# B&R Automation Studio project Parker_BMM_ST_V5_3147_V12
Automation Studio 4.2.12.129 SP

## Configuration 5AP1180_1505_parker3147

CPU 5PPC2100.BY01-000, AutomationRuntime D4.26, Build 4.1.2, Vc V4.26.8, Safety 0.0

### Task classes (Cpu.sw)
```
Cyclic#1 (cycle 2000 us, tolerance 0 us):
  tk1_in <- In_Out.tk1_in.prg
  timer <- process.timer.prg
  clamp <- process.clamp.prg
  carriage <- process.carriage.prg
  blowpin <- process.blowpin.prg
  blowpin2 <- process.blowpin2.prg
  extrlift <- process.extrlift.prg
  mc_pwr <- Motion.mc_pwr.prg [disabled]
  tk1_out <- In_Out.tk1_out.prg
  parison <- thickness.parison.prg
  robot <- process.robot.prg
  r_carriage <- Motion.r_carriage.prg [disabled]
  l_carriage <- Motion.l_carriage.prg [disabled]
  r_blowpin <- Motion.r_blowpin.prg [disabled]
  l_blowpin <- Motion.l_blowpin.prg [disabled]
  r_blowpin2 <- Motion.r_blowpin2.prg [disabled]
  l_blowpin2 <- Motion.l_blowpin2.prg [disabled]
  l_clamp <- Motion.l_clamp.prg [disabled]
  r_clamp <- Motion.r_clamp.prg [disabled]
  l_transfer <- Motion.l_transfer.prg [disabled]
  r_transfer <- Motion.r_transfer.prg [disabled]
  mc_extrlif <- Motion.mc_extrlift.prg [disabled]
  mc_thick <- Motion.mc_thick.prg [disabled]
  Trace <- screen.Trace.prg
  clean_Test <- (binary)
Cyclic#2 (cycle 10000 us, tolerance 100000 us):
  h_pwm <- Heating.h_pwm.prg
  tk2_io <- In_Out.tk2_io.prg
Cyclic#3 (cycle 4000 us, tolerance 100000 us):
  cutter <- process.cutter.prg
  cutneck <- process.cutneck.prg
  cooldef <- process.cooldef.prg
  blowdef <- process.blowdef.prg
  bdeflash <- process.bdeflash.prg
  tdeflash <- process.tdeflash.prg
  pullbottom <- process.pullbottom.prg
  inerpin <- process.inerpin.prg
  highblow <- process.highblow.prg
  lowblow <- process.lowblow.prg
  hookpin <- process.hookpin.prg
  coolpin <- process.coolpin.prg
  coolpin2 <- process.coolpin2.prg
  coolpin3 <- process.coolpin3.prg
  coolblw <- process.coolblw.prg
  coolblw2 <- process.coolblw2.prg
  coolblw3 <- process.coolblw3.prg
  robotopncl <- process.robotopncls.prg
  submold <- process.submold.prg
  pinpart <- process.pinpart.prg
  screw <- process.screw.prg
  sealer <- process.sealer.prg
  bblowpin <- process.bblowpin.prg
  support <- process.support.prg
  tonnage <- process.tonnage.prg
  autorun <- process.autorun.prg
  extru_plk <- machine.extru_plk.prg [disabled]
  extruder <- machine.extruder.prg [disabled]
  extruder_M <- machine.extruder_Mix.prg
  Acs580Ctl <- machine.Acs580Ctl.prg
  plate <- process.plate.prg
Cyclic#4 (cycle 20000 us, tolerance 200000 us):
  keyled <- screen.keyled.prg
  manual <- machine.manual.prg
  calib <- machine.calib.prg
  reset <- machine.reset.prg
  workmode <- machine.workmode.prg
  mode <- machine.mode.prg
  panel <- screen.panel.prg
  hmi_cpy <- screen.hmi_cpy.prg
  pump <- machine.pump.prg
  mac_lubr <- machine.mac_lubr.prg
  oil_accu <- machine.oil_accu.prg
  mbusMaster <- comm.mbusMaster.prg
  clean <- machine.clean.prg
  length <- process.length.prg
Cyclic#5 (cycle 500000 us, tolerance 500000 us):
  h_pid <- Heating.h_pid.prg
Cyclic#6 (cycle 30000 us, tolerance 3000000 us):
  cur_cal <- thickness.cur_cal.prg
  exchange <- thickness.exchange.prg
Cyclic#7 (cycle 50000 us, tolerance 5000000 us):
  cur_edit <- thickness.cur_edit.prg
  cur_draw <- thickness.cur_draw.prg
  pvchg <- VarChgLog.pvchg.prg
Cyclic#8 (cycle 200000 us, tolerance 30000000 us):
  spc_ctrl <- spc.spc_ctrl.prg
  trend <- Heating.trend.prg
  h_plan <- Heating.h_plan.prg
  scrshot <- screen.scrshot.prg
  hmiset <- screen.hmiset.prg
  password <- screen.password.prg
  modem <- comm.modem.prg
  vpn <- screen.vpn.prg
  recipe <- recipeMan.recipe.prg
  multsave <- recipeMan.multsave.prg
  oncesave <- recipeMan.oncesave.prg
  cur_save <- thickness.cur_save.prg
  cfg_cpy <- recipeMan.cfg_cpy.prg
  alarm <- machine.alarm.prg
  energy <- machine.energy.prg
  epl <- comm.epl.prg
DataObjects: mb_cmd <- comm.mb_cmd.dob, var_fix <- recipeMan.var_fix.dob, var_mold <- recipeMan.var_mold.dob, log_txt <- log_info.log_txt.dob, pv_chg <- VarChgLog.pv_chg.dob, cfg_dat <- recipeMan.cfg_dat.dob, Acp10sys, recName, recFix, recCurve, recMold
NcDataObjects: TransferR <- Motion.init.TransferR.dob, CarriageR <- Motion.init.CarriageR.dob, CarriageL <- Motion.init.CarriageL.dob, BlowPinR <- Motion.init.BlowPinR.dob, BlowPinL <- Motion.init.BlowPinL.dob, BlowPin2R <- Motion.init.BlowPin2R.dob, BlowPin2L <- Motion.init.BlowPin2L.dob, ThickInit <- Motion.init.ThickInit.dob, Tansfer <- Motion.para.Tansfer.dob, UpDn <- Motion.para.UpDn.dob, CarraigeLR <- Motion.para.CarraigeLR.dob, BlowPinLR <- Motion.para.BlowPinLR.dob, nCarraigeL <- Motion.para.nCarraigeLR.dob, nBlowPinLR <- Motion.para.nBlowPinLR.dob, BlowPin2LR <- Motion.para.BlowPin2LR.dob, ClampLR <- Motion.para.ClampLR.dob, acp10etxen <- Motion.acp10etxen.dob, Power <- Motion.init.Power.dob, Power1 <- Motion.para.Power.dob, ClampR <- Motion.init.ClampR.dob, ClampL <- Motion.init.ClampL.dob, ExtrLift1 <- Motion.init.ExtrLift.dob, ExtrLift2 <- Motion.para.ExtrLift.dob, ThickPara <- Motion.para.ThickPara.dob, 0804Thick, 0129_C2, gAxisPwri, gAxisPwra
VcDataObjects: visu15 <- Visu.visu15.dob
Binaries: TCData, vctcal, vccnum, vccalarm, vccovl, vcshared, visu1502, vcfile, vccstr, vccline, arial, vcctrend, vcchtml, vcgclass, vccbtn, vcrt, vccdbox, visu1503, vcclbox, simsun, vcctext, vccbmp, vcfntttf, vcalarm, vcdsint, visu1501, vccshape, vcchspot, vcmgr, vcdsloc, visvc, vccurl, vccdt, vccbar, vcpdsw, vcxml, vccscale, vcbclass, vcnet, vcpdvnc, vccddbox, vccpopup, timesbd, times, arialxsr, vccslider, vcpfar00, Role, ashwd, arconfig, iomap, User, asfw, sysconf, Acp10map, acp10cfg, vcpfmtcx, vcpk, vcpfapc, vcptelo, vcpdi815, vcpdi855, vcpdihd, vcpkat, tahomabd, arialbd, tahoma, myxh_1, myxh
Libraries: visapi, FileIO, runtime, sys_lib, standard, operator, dvframe, DataObj, Convert, brsystem, astime, asstring, AsIO, AsArLog, AsARCfg, Motorky, DRV_mbus, LoopConR, SimpFun, HydCtrl, NcGlobal, Acp10par, Acp10_MC, AsHydCon, AsEPL, Acp10man, Acp10sim, vcscrsht, powerlnk, vcresman
```

### Hardware
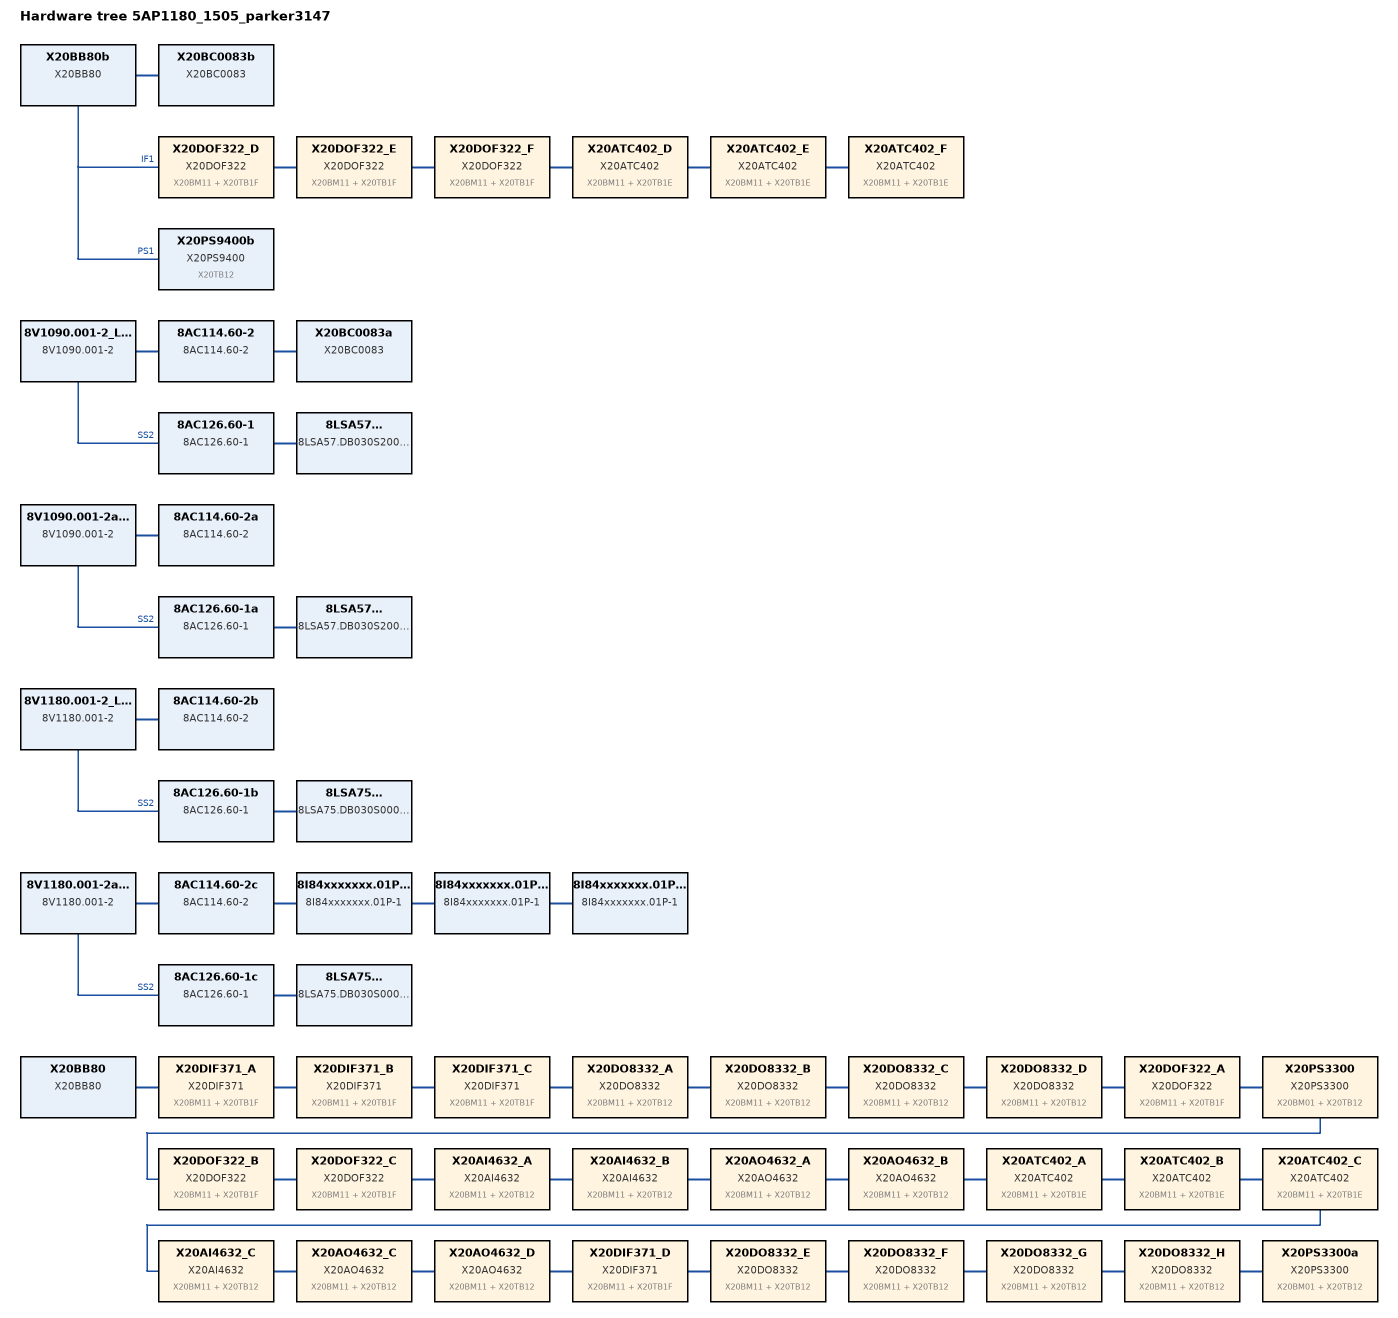
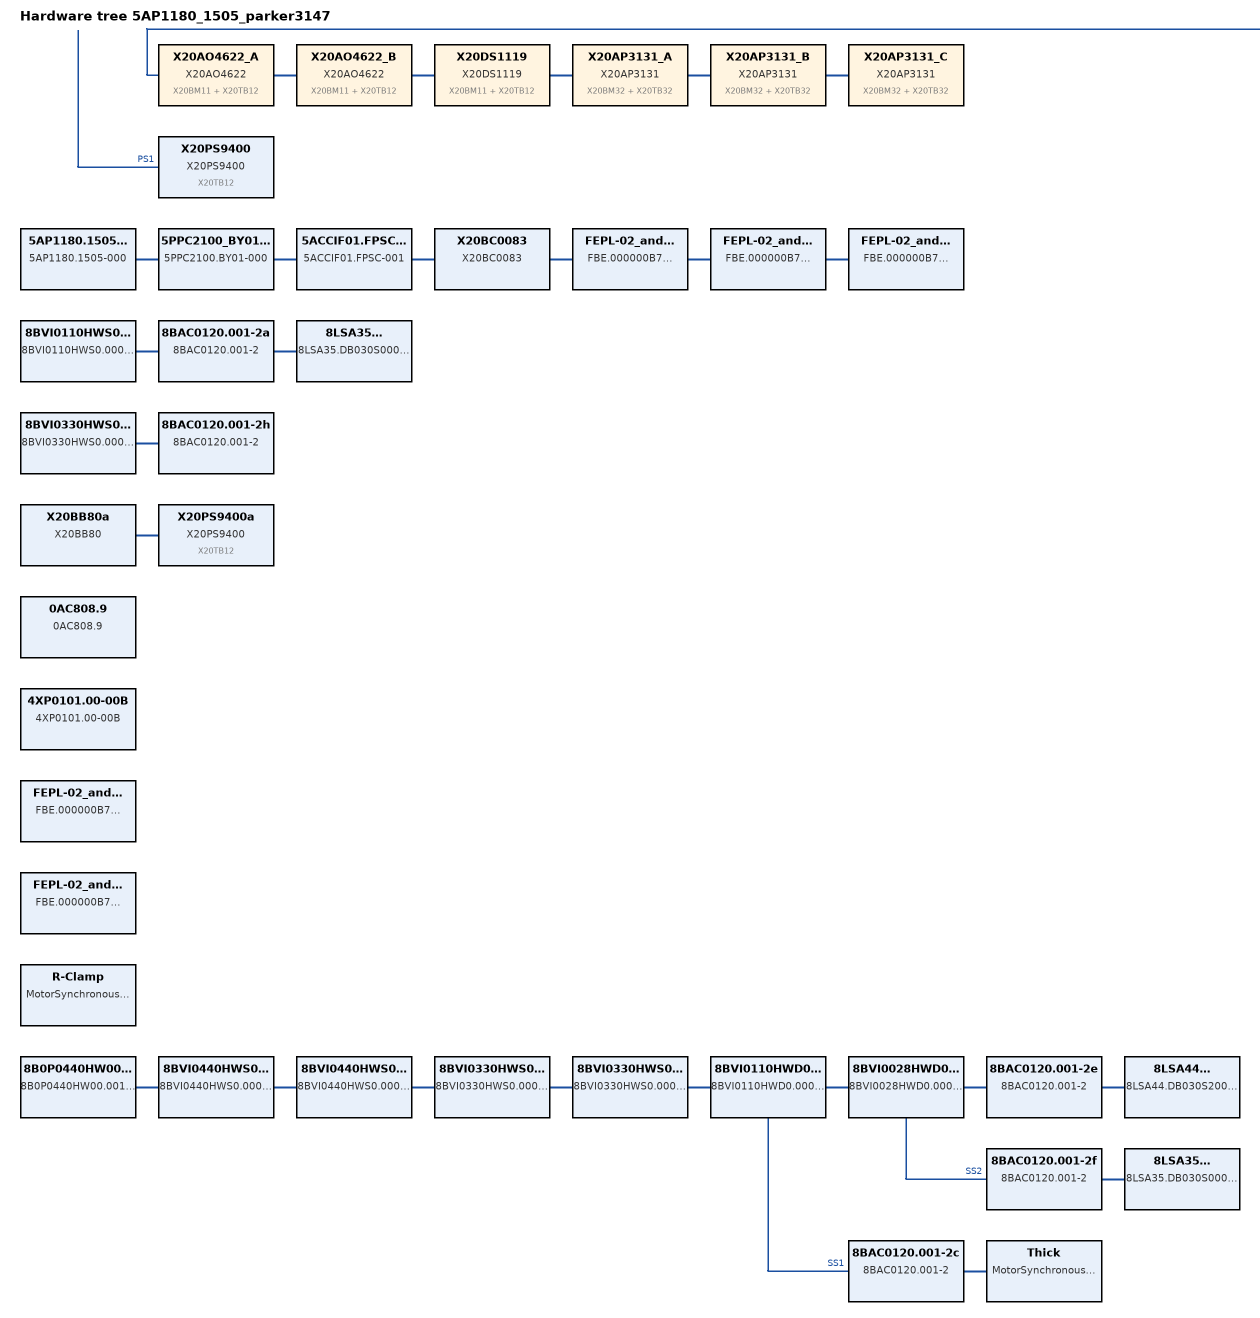
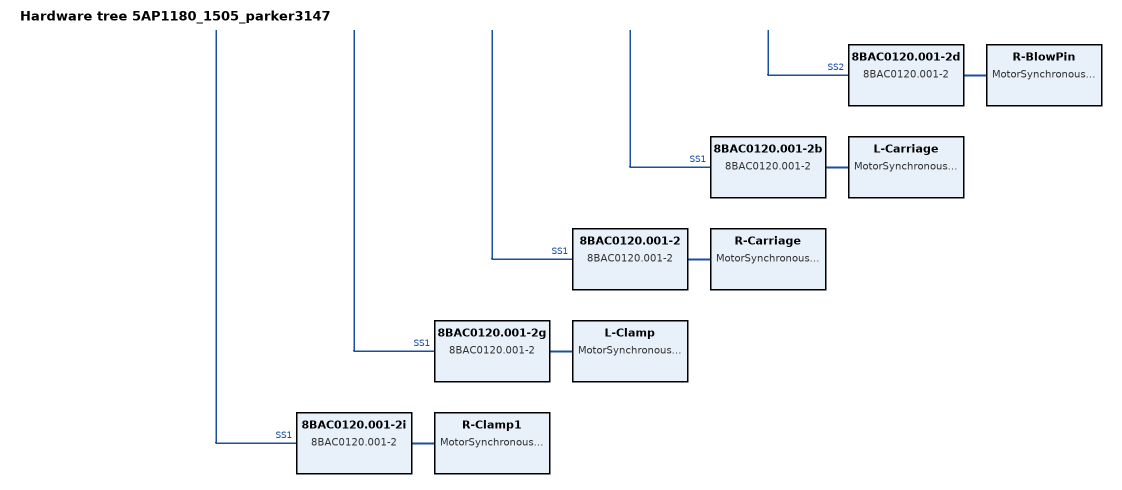
```
0AC808.9 : 0AC808.9 v1.0.0.0
4XP0101.00-00B : 4XP0101.00-00B v2.1.0.0
  Supervision = off
5ACCIF01.FPSC-001 : 5ACCIF01.FPSC-001 v1.8.1.0  [SL -> 5PPC2100_BY01_000.SL1]
5AP1180.1505-000 : 5AP1180.1505-000 v2.0.0.0
  VcObjectName = visu15
5PPC2100_BY01_000 : 5PPC2100.BY01-000 v1.4.0.0  [SY -> 5AP1180.1505-000.SY1]
  Connector IF3:
    ActivateDevice = 1
    Mode = Manual
    InternetAddress = 10.86.100.212
    SubnetMask = 255.255.255.0
    InaNodeNumber = 1
    Vnc1
    VncVcObjectName1 = visu15
    VncMaxConnections1 = 2
  Connector IF4:
    ActivateDevice = 1
    Mode = Manual
    InternetAddress = 192.168.1.100
    SubnetMask = 255.255.255.0
  ConfigurationID = bmm_5AP1180_1505_000
  UserRamDevice = PCI.1.PPC21xx.SRAM
  UserRamSize = 260864
  RemMemDevice = PCI.1.PPC21xx.SRAM
  RemMemSize = 262144
  PermanentPvSize = 12000
  RemanentGlobalPvSize = 20000
  VolatileGlobalPvSize = 200000
  EnableUsbRemoteInstall = 1
  TimerDeviceType = EPLX2X
  TimerDevice = 5ACCIF01.FPSC-001.IF1
  TaskClassIdleTime = 2000
  Cyclic1Duration = 2000
  Cyclic1Tolerance = 0
  Cyclic1Stack = 8192
  Cyclic1Output = 1
  Cyclic2Duration = 10000
  Cyclic2Tolerance = 100000
  Cyclic2Stack = 8192
  Cyclic3Duration = 4000
  Cyclic3Tolerance = 100000
  Cyclic3Stack = 8192
  Cyclic4Duration = 20000
  Cyclic4Tolerance = 200000
  Cyclic4Stack = 8192
  Cyclic5Duration = 500000
  Cyclic5Tolerance = 500000
  Cyclic5Stack = 20000
  Cyclic6Duration = 30000
  Cyclic6Tolerance = 3000000
  Cyclic6Stack = 8192
  Cyclic7Duration = 50000
  Cyclic7Tolerance = 5000000
  Cyclic7Stack = 8192
  Cyclic8Duration = 200000
  Cyclic8Tolerance = 30000000
  Cyclic8Stack = 30000
  FileDevice1
  FileDeviceName1 = USB_1
  FileDevicePath1 = /bd0
  FileDevice2
  FileDeviceName2 = USB_2
  FileDevicePath2 = /bd16
  FileDevice3
  FileDeviceName3 = SCREEN_1
  FileDevicePath3 = /bd0\\ScreenShot
  FileDevice4
  FileDeviceName4 = SCREEN_2
  FileDevicePath4 = /bd16\\ScreenShot
  FileDevice5
  FileDeviceName5 = SINGLE_1
  FileDevicePath5 = /bd0\\SingleRecipe
  FileDevice6
  FileDeviceName6 = SINGLE_2
  FileDevicePath6 = /bd16\\SingleRecipe
  FileDevice7
  FileDeviceName7 = ALL_1
  FileDevicePath7 = /bd0\\AllRecipe
  FileDevice8
  FileDeviceName8 = ALL_2
  FileDevicePath8 = /bd16\\AllRecipe
  FileDevice9
  FileDeviceName9 = USER
  FileDevicePath9 = F:\
  FileDevice10
  FileDeviceName10 = DOC
  FileDevicePath10 = C:\AR000\C
  TimeZone = 315
8AC114.60-2 : 8AC114.60-2 v1.0.0.8 (Disabled=true)  [SS -> 8V1090.001-2_L_BlowPin.SS1; PLK1 -> X20BC0083a.PLK2 (NodeNumber=3); PLK2 -> 8AC114.60-2a.PLK1 (NodeNumber=3)]
8AC114.60-2a : 8AC114.60-2 v1.0.0.8 (Disabled=true)  [SS -> 8V1090.001-2a_R_BlowPin.SS1; PLK1 -> 8AC114.60-2.PLK2 (NodeNumber=4); PLK2 -> 8AC114.60-2b.PLK1 (NodeNumber=4)]
8AC114.60-2b : 8AC114.60-2 v1.0.0.8 (Disabled=true)  [SS -> 8V1180.001-2_L_Carriage.SS1; PLK1 -> 8AC114.60-2a.PLK2 (NodeNumber=5); PLK2 -> 8AC114.60-2c.PLK1 (NodeNumber=5)]
8AC114.60-2c : 8AC114.60-2 v1.0.0.8 (Disabled=true)  [SS -> 8V1180.001-2a_R_Carriage.SS1; PLK1 -> 8AC114.60-2b.PLK2 (NodeNumber=6); PLK2 -> 8I84xxxxxxx.01P-1b.PLK1 (NodeNumber=6)]
8AC126.60-1 : 8AC126.60-1 v2.2.0.0 (Disabled=true)  [SS -> 8V1090.001-2_L_BlowPin.SS2]
8AC126.60-1a : 8AC126.60-1 v2.2.0.0 (Disabled=true)  [SS -> 8V1090.001-2a_R_BlowPin.SS2]
8AC126.60-1b : 8AC126.60-1 v2.2.0.0 (Disabled=true)  [SS -> 8V1180.001-2_L_Carriage.SS2]
8AC126.60-1c : 8AC126.60-1 v2.2.0.0 (Disabled=true)  [SS -> 8V1180.001-2a_R_Carriage.SS2]
8B0P0440HW00.001-1 : 8B0P0440HW00.001-1 v1.0.0.4  [PLK2 -> 8BVI0440HWS0.000-1.PLK1 (NodeNumber=3)]
  BothEndSwitchesAreNormallyOpen_r1 = on
  QuickStopIsNormallyOpen_r1 = on
8BAC0120.001-2 : 8BAC0120.001-2 v2.2.0.0 (Disabled=true)  [SS -> 8BVI0330HWS0.000-1.SS1]
8BAC0120.001-2a : 8BAC0120.001-2 v2.2.0.0 (Disabled=true)  [SS -> 8BVI0110HWS0.000-1.SS1]
8BAC0120.001-2b : 8BAC0120.001-2 v2.2.0.0 (Disabled=true)  [SS -> 8BVI0330HWS0.000-1a.SS1]
8BAC0120.001-2c : 8BAC0120.001-2 v2.2.0.0  [SS -> 8BVI0110HWD0.000-1.SS1]
8BAC0120.001-2d : 8BAC0120.001-2 v2.2.0.0  [SS -> 8BVI0110HWD0.000-1.SS2]
8BAC0120.001-2e : 8BAC0120.001-2 v2.2.0.0 (Disabled=true)  [SS -> 8BVI0028HWD0.000-1.SS1]
8BAC0120.001-2f : 8BAC0120.001-2 v2.2.0.0 (Disabled=true)  [SS -> 8BVI0028HWD0.000-1.SS2]
8BAC0120.001-2g : 8BAC0120.001-2 v2.2.0.0 (Disabled=true)  [SS -> 8BVI0440HWS0.000-1a.SS1]
8BAC0120.001-2h : 8BAC0120.001-2 v2.2.0.0 (Disabled=true)  [SS -> 8BVI0330HWS0.000-1b.SS1]
8BAC0120.001-2i : 8BAC0120.001-2 v2.2.0.0 (Disabled=true)  [SS -> 8BVI0440HWS0.000-1.SS1]
8BVI0028HWD0.000-1 : 8BVI0028HWD0.000-1 v2.3.0.1 (Disabled=true)  [PLK1 -> 8BVI0110HWD0.000-1.PLK2 (NodeNumber=12); MT2 -> 8LSA35.DB030S000-3a.MT]
  PowerSupply = passive
8BVI0110HWD0.000-1 : 8BVI0110HWD0.000-1 v2.3.0.1  [PLK1 -> 8BVI0330HWS0.000-1a.PLK2 (NodeNumber=11); PLK2 -> 8BVI0028HWD0.000-1.PLK1 (NodeNumber=11); MT2 -> R-BlowPin.MT]
  PowerSupply = passive
8BVI0110HWS0.000-1 : 8BVI0110HWS0.000-1 v1.0.0.4 (Disabled=true)
  PowerSupply = passive
  FunctionModel = SingleAxis
8BVI0330HWS0.000-1 : 8BVI0330HWS0.000-1 v2.3.0.1 (Disabled=true)  [PLK1 -> 8BVI0440HWS0.000-1a.PLK2 (NodeNumber=9); PLK2 -> 8BVI0330HWS0.000-1a.PLK1 (NodeNumber=9)]
  PowerSupply = passive
  FunctionModel = SingleAxis
8BVI0330HWS0.000-1a : 8BVI0330HWS0.000-1 v2.3.0.1 (Disabled=true)  [PLK1 -> 8BVI0330HWS0.000-1.PLK2 (NodeNumber=10); PLK2 -> 8BVI0110HWD0.000-1.PLK1 (NodeNumber=10)]
  PowerSupply = passive
  FunctionModel = SingleAxis
8BVI0330HWS0.000-1b : 8BVI0330HWS0.000-1 v2.3.0.1 (Disabled=true)
  PowerSupply = passive
  FunctionModel = SingleAxis
8BVI0440HWS0.000-1 : 8BVI0440HWS0.000-1 v1.0.0.4 (Disabled=true)  [PLK1 -> 8B0P0440HW00.001-1.PLK2 (NodeNumber=7); PLK2 -> 8BVI0440HWS0.000-1a.PLK1 (NodeNumber=7)]
8BVI0440HWS0.000-1a : 8BVI0440HWS0.000-1 v1.0.0.4 (Disabled=true)  [PLK1 -> 8BVI0440HWS0.000-1.PLK2 (NodeNumber=8); PLK2 -> 8BVI0330HWS0.000-1.PLK1 (NodeNumber=8)]
8I84xxxxxxx.01P-1 : 8I84xxxxxxx.01P-1 v1.0.9.2 (Disabled=true)  [PLK1 -> 8I84xxxxxxx.01P-1b.PLK2 (NodeNumber=8); PLK2 -> 8I84xxxxxxx.01P-1a.PLK1 (NodeNumber=8)]
  FunctionModel = Standard
  Supervision = off
  ACC = 150
  DEC = 150
  AC2 = 150
  DE2 = 150
  ITH = 1399
  NPR = 7500
  UNS = 380
  NCR = 1399
  NSP = 1480
  PTCL = 1
8I84xxxxxxx.01P-1a : 8I84xxxxxxx.01P-1 v1.0.9.2 (Disabled=true)  [PLK1 -> 8I84xxxxxxx.01P-1.PLK2 (NodeNumber=9)]
  FunctionModel = Standard
  Supervision = off
  ACC = 150
  DEC = 150
  AC2 = 150
  DE2 = 150
  ITH = 580
  NPR = 3000
  UNS = 380
  NCR = 580
  NSP = 1475
  PTCL = 1
8I84xxxxxxx.01P-1b : 8I84xxxxxxx.01P-1 v1.0.9.2 (Disabled=true)  [PLK1 -> 8AC114.60-2c.PLK2 (NodeNumber=7); PLK2 -> 8I84xxxxxxx.01P-1.PLK1 (NodeNumber=7)]
  FunctionModel = Standard
  Supervision = off
  ACC = 150
  DEC = 150
  AC2 = 150
  DE2 = 150
  ITH = 580
  NPR = 3000
  UNS = 380
  NCR = 580
  NSP = 1475
  PTCL = 1
8LSA35.DB030S000-3 : 8LSA35.DB030S000-3 v1.0.2.34 (Disabled=true)  [EC -> 8BAC0120.001-2a.EC; MT -> 8BVI0110HWS0.000-1.MT1]
  MOTOR_TYPE = 16#0004
  MOTOR_COMPATIBILITY = 16#0207
  MOTOR_WIND_CONNECT = 1
  MOTOR_BRAKE_TYPE = 0
  MOTOR_BRAKE_CURR_RATED = 0
  MOTOR_BRAKE_TORQ_RATED = 0
  MOTOR_BRAKE_ON_TIME = 0
  MOTOR_BRAKE_OFF_TIME = 0
  MOTOR_BRAKE_RESISTANCE = 0
  MOTOR_BRAKE_INDUCTANCE = 0
  MOTOR_BRAKE_VOLT_REL = 0
  MOTOR_BRAKE_VOLT_HOLD = 0
  MOTOR_BRAKE_VOLT_MAX = 0
  MOTOR_TEMPSENS_PAR1 = 31
  MOTOR_TEMPSENS_PAR2 = 289
  MOTOR_TEMPSENS_PAR3 = -30
  MOTOR_TEMPSENS_PAR4 = -0.65
  MOTOR_TEMPSENS_PAR5 = 29.06
  MOTOR_TEMPSENS_PAR6 = 58.83
  MOTOR_TEMPSENS_PAR7 = 88.17
  MOTOR_TEMPSENS_PAR8 = 117.42
  MOTOR_TEMPSENS_PAR9 = 147.14
  MOTOR_TEMPSENS_PAR10 = 175
  MOTOR_TEMPSENS_TYPE = 4353
  MOTOR_TEMPSENS_LIM = 130
  MOTOR_POLEPAIRS = 4
  MOTOR_VOLTAGE_RATED = 400
  MOTOR_VOLTAGE_CONST = 87.96
  MOTOR_SPEED_RATED = 3000
  MOTOR_SPEED_MAX = 9000
  MOTOR_TORQ_STALL = 2.3
  MOTOR_TORQ_RATED = 2.1
  MOTOR_TORQ_MAX = 9.2
  MOTOR_TORQ_CONST = 1.45
  MOTOR_CURR_STALL = 1.6
  MOTOR_CURR_RATED = 1.4
  MOTOR_CURR_MAX = 6.8
  MOTOR_WIND_CROSS_SECT = 0.181
  MOTOR_STATOR_RESISTANCE = 12.22
  MOTOR_STATOR_INDUCTANCE = 0.063
  MOTOR_INERTIA = 9E-05
  MOTOR_COMMUT_OFFSET = 1000000
  MOTOR_WIND_TEMP_MAX = 110
  MOTOR_TAU_THERM = 2040
  MOTOR_AMB_TEMP_RATED = 40
  MOTOR_TEMPMODEL_REFSENS = 0
  MOTOR_TEMPMODEL_RES1 = 0
  MOTOR_TEMPMODEL_CAP1 = 0
  MOTOR_TEMPMODEL_RES2 = 0
  MOTOR_TEMPMODEL_CAP2 = 0
  MOTOR_TEMPMODEL_LOSS1 = 0
  MOTOR_TEMPMODEL_LOSS2 = 0
  MOTOR_TEMPMODEL_MODE = 16#FFFF
  MOTOR_ENCOD_TEMP_LIM = 120
8LSA35.DB030S000-3a : 8LSA35.DB030S000-3 v1.0.2.34 (Disabled=true)  [EC -> 8BAC0120.001-2f.EC; MT -> 8BVI0028HWD0.000-1.MT2]
  MOTOR_TYPE = 16#0004
  MOTOR_COMPATIBILITY = 16#0207
  MOTOR_WIND_CONNECT = 1
  MOTOR_BRAKE_TYPE = 0
  MOTOR_BRAKE_CURR_RATED = 0
  MOTOR_BRAKE_TORQ_RATED = 0
  MOTOR_BRAKE_ON_TIME = 0
  MOTOR_BRAKE_OFF_TIME = 0
  MOTOR_BRAKE_RESISTANCE = 0
  MOTOR_BRAKE_INDUCTANCE = 0
  MOTOR_BRAKE_VOLT_REL = 0
  MOTOR_BRAKE_VOLT_HOLD = 0
  MOTOR_BRAKE_VOLT_MAX = 0
  MOTOR_TEMPSENS_PAR1 = 31
  MOTOR_TEMPSENS_PAR2 = 289
  MOTOR_TEMPSENS_PAR3 = -30
  MOTOR_TEMPSENS_PAR4 = -0.65
  MOTOR_TEMPSENS_PAR5 = 29.06
  MOTOR_TEMPSENS_PAR6 = 58.83
  MOTOR_TEMPSENS_PAR7 = 88.17
  MOTOR_TEMPSENS_PAR8 = 117.42
  MOTOR_TEMPSENS_PAR9 = 147.14
  MOTOR_TEMPSENS_PAR10 = 175
  MOTOR_TEMPSENS_TYPE = 4353
  MOTOR_TEMPSENS_LIM = 130
  MOTOR_POLEPAIRS = 4
  MOTOR_VOLTAGE_RATED = 400
  MOTOR_VOLTAGE_CONST = 87.96
  MOTOR_SPEED_RATED = 3000
  MOTOR_SPEED_MAX = 9000
  MOTOR_TORQ_STALL = 2.3
  MOTOR_TORQ_RATED = 2.1
  MOTOR_TORQ_MAX = 9.2
  MOTOR_TORQ_CONST = 1.45
  MOTOR_CURR_STALL = 1.6
  MOTOR_CURR_RATED = 1.4
  MOTOR_CURR_MAX = 6.8
  MOTOR_WIND_CROSS_SECT = 0.181
  MOTOR_STATOR_RESISTANCE = 12.22
  MOTOR_STATOR_INDUCTANCE = 0.063
  MOTOR_INERTIA = 9E-05
  MOTOR_COMMUT_OFFSET = 1000000
  MOTOR_WIND_TEMP_MAX = 110
  MOTOR_TAU_THERM = 2040
  MOTOR_AMB_TEMP_RATED = 40
  MOTOR_TEMPMODEL_REFSENS = 0
  MOTOR_TEMPMODEL_RES1 = 0
  MOTOR_TEMPMODEL_CAP1 = 0
  MOTOR_TEMPMODEL_RES2 = 0
  MOTOR_TEMPMODEL_CAP2 = 0
  MOTOR_TEMPMODEL_LOSS1 = 0
  MOTOR_TEMPMODEL_LOSS2 = 0
  MOTOR_TEMPMODEL_MODE = 16#FFFF
  MOTOR_ENCOD_TEMP_LIM = 120
8LSA44.DB030S200-3 : 8LSA44.DB030S200-3 v1.0.8.37 (Disabled=true)  [EC -> 8BAC0120.001-2e.EC; MT -> 8BVI0028HWD0.000-1.MT1]
  MOTOR_TYPE = 16#0002
  MOTOR_COMPATIBILITY = 16#0207
  MOTOR_WIND_CONNECT = 1
  MOTOR_BRAKE_TYPE = 16#FFFF
  MOTOR_BRAKE_CURR_RATED = 0.75
  MOTOR_BRAKE_TORQ_RATED = 8
  MOTOR_BRAKE_ON_TIME = 0.038
  MOTOR_BRAKE_OFF_TIME = 0.055
  MOTOR_BRAKE_RESISTANCE = 0
  MOTOR_BRAKE_INDUCTANCE = 0
  MOTOR_BRAKE_VOLT_REL = 0
  MOTOR_BRAKE_VOLT_HOLD = 0
  MOTOR_BRAKE_VOLT_MAX = 0
  MOTOR_TEMPSENS_PAR1 = 31
  MOTOR_TEMPSENS_PAR2 = 289
  MOTOR_TEMPSENS_PAR3 = -30
  MOTOR_TEMPSENS_PAR4 = -0.65
  MOTOR_TEMPSENS_PAR5 = 29.06
  MOTOR_TEMPSENS_PAR6 = 58.83
  MOTOR_TEMPSENS_PAR7 = 88.17
  MOTOR_TEMPSENS_PAR8 = 117.42
  MOTOR_TEMPSENS_PAR9 = 147.14
  MOTOR_TEMPSENS_PAR10 = 175
  MOTOR_TEMPSENS_TYPE = 4353
  MOTOR_TEMPSENS_LIM = 130
  MOTOR_POLEPAIRS = 5
  MOTOR_VOLTAGE_RATED = 400
  MOTOR_VOLTAGE_CONST = 98.44
  MOTOR_SPEED_RATED = 3000
  MOTOR_SPEED_MAX = 12000
  MOTOR_TORQ_STALL = 6
  MOTOR_TORQ_RATED = 4.62
  MOTOR_TORQ_MAX = 22.8
  MOTOR_TORQ_CONST = 1.63
  MOTOR_CURR_STALL = 3.7
  MOTOR_CURR_RATED = 2.8
  MOTOR_CURR_MAX = 21.9
  MOTOR_WIND_CROSS_SECT = 0.503
  MOTOR_STATOR_RESISTANCE = 3.6
  MOTOR_STATOR_INDUCTANCE = 0.024
  MOTOR_INERTIA = 0.000327
  MOTOR_COMMUT_OFFSET = 1000000
  MOTOR_WIND_TEMP_MAX = 110
  MOTOR_TAU_THERM = 1800
  MOTOR_AMB_TEMP_RATED = 40
  MOTOR_TEMPMODEL_REFSENS = 0
  MOTOR_TEMPMODEL_RES1 = 0
  MOTOR_TEMPMODEL_CAP1 = 0
  MOTOR_TEMPMODEL_RES2 = 0
  MOTOR_TEMPMODEL_CAP2 = 0
  MOTOR_TEMPMODEL_LOSS1 = 0
  MOTOR_TEMPMODEL_LOSS2 = 0
  MOTOR_TEMPMODEL_MODE = 16#FFFF
  MOTOR_ENCOD_TEMP_LIM = 120
8LSA57.DB030S200-3 : 8LSA57.DB030S200-3 v2.2.0.1 (Disabled=true)  [EC -> 8AC126.60-1.EC; MT -> 8V1090.001-2_L_BlowPin.MT1]
  MOTOR_TYPE = 16#0002
  MOTOR_COMPATIBILITY = 16#0207
  MOTOR_WIND_CONNECT = 1
  MOTOR_BRAKE_TYPE = 16#FFFF
  MOTOR_BRAKE_CURR_RATED = 1
  MOTOR_BRAKE_TORQ_RATED = 15
  MOTOR_BRAKE_ON_TIME = 0.01
  MOTOR_BRAKE_OFF_TIME = 0.05
  MOTOR_BRAKE_RESISTANCE = 0
  MOTOR_BRAKE_INDUCTANCE = 0
  MOTOR_BRAKE_VOLT_REL = 0
  MOTOR_BRAKE_VOLT_HOLD = 0
  MOTOR_BRAKE_VOLT_MAX = 0
  MOTOR_TEMPSENS_PAR1 = 31
  MOTOR_TEMPSENS_PAR2 = 289
  MOTOR_TEMPSENS_PAR3 = -30
  MOTOR_TEMPSENS_PAR4 = -0.65
  MOTOR_TEMPSENS_PAR5 = 29.06
  MOTOR_TEMPSENS_PAR6 = 58.83
  MOTOR_TEMPSENS_PAR7 = 88.17
  MOTOR_TEMPSENS_PAR8 = 117.42
  MOTOR_TEMPSENS_PAR9 = 147.14
  MOTOR_TEMPSENS_PAR10 = 175
  MOTOR_TEMPSENS_TYPE = 4353
  MOTOR_TEMPSENS_LIM = 130
  MOTOR_POLEPAIRS = 4
  MOTOR_VOLTAGE_RATED = 400
  MOTOR_VOLTAGE_CONST = 98.44
  MOTOR_SPEED_RATED = 3000
  MOTOR_SPEED_MAX = 9000
  MOTOR_TORQ_STALL = 20
  MOTOR_TORQ_RATED = 17.5
  MOTOR_TORQ_MAX = 69
  MOTOR_TORQ_CONST = 1.63
  MOTOR_CURR_STALL = 12.3
  MOTOR_CURR_RATED = 10.7
  MOTOR_CURR_MAX = 52.6
  MOTOR_WIND_CROSS_SECT = 2.01
  MOTOR_STATOR_RESISTANCE = 0.62
  MOTOR_STATOR_INDUCTANCE = 0.00721
  MOTOR_INERTIA = 0.00148
  MOTOR_COMMUT_OFFSET = 1000000
  MOTOR_WIND_TEMP_MAX = 110
  MOTOR_TAU_THERM = 2760
  MOTOR_AMB_TEMP_RATED = 40
  MOTOR_TEMPMODEL_REFSENS = 0
  MOTOR_TEMPMODEL_RES1 = 0
  MOTOR_TEMPMODEL_CAP1 = 0
  MOTOR_TEMPMODEL_RES2 = 0
  MOTOR_TEMPMODEL_CAP2 = 0
  MOTOR_TEMPMODEL_LOSS1 = 0
  MOTOR_TEMPMODEL_LOSS2 = 0
  MOTOR_TEMPMODEL_MODE = 16#FFFF
  MOTOR_ENCOD_TEMP_LIM = 120
8LSA57.DB030S200-3a : 8LSA57.DB030S200-3 v2.2.0.1 (Disabled=true)  [EC -> 8AC126.60-1a.EC; MT -> 8V1090.001-2a_R_BlowPin.MT1]
  MOTOR_TYPE = 16#0002
  MOTOR_COMPATIBILITY = 16#0207
  MOTOR_WIND_CONNECT = 1
  MOTOR_BRAKE_TYPE = 16#FFFF
  MOTOR_BRAKE_CURR_RATED = 1
  MOTOR_BRAKE_TORQ_RATED = 15
  MOTOR_BRAKE_ON_TIME = 0.01
  MOTOR_BRAKE_OFF_TIME = 0.05
  MOTOR_BRAKE_RESISTANCE = 0
  MOTOR_BRAKE_INDUCTANCE = 0
  MOTOR_BRAKE_VOLT_REL = 0
  MOTOR_BRAKE_VOLT_HOLD = 0
  MOTOR_BRAKE_VOLT_MAX = 0
  MOTOR_TEMPSENS_PAR1 = 31
  MOTOR_TEMPSENS_PAR2 = 289
  MOTOR_TEMPSENS_PAR3 = -30
  MOTOR_TEMPSENS_PAR4 = -0.65
  MOTOR_TEMPSENS_PAR5 = 29.06
  MOTOR_TEMPSENS_PAR6 = 58.83
  MOTOR_TEMPSENS_PAR7 = 88.17
  MOTOR_TEMPSENS_PAR8 = 117.42
  MOTOR_TEMPSENS_PAR9 = 147.14
  MOTOR_TEMPSENS_PAR10 = 175
  MOTOR_TEMPSENS_TYPE = 4353
  MOTOR_TEMPSENS_LIM = 130
  MOTOR_POLEPAIRS = 4
  MOTOR_VOLTAGE_RATED = 400
  MOTOR_VOLTAGE_CONST = 98.44
  MOTOR_SPEED_RATED = 3000
  MOTOR_SPEED_MAX = 9000
  MOTOR_TORQ_STALL = 20
  MOTOR_TORQ_RATED = 17.5
  MOTOR_TORQ_MAX = 69
  MOTOR_TORQ_CONST = 1.63
  MOTOR_CURR_STALL = 12.3
  MOTOR_CURR_RATED = 10.7
  MOTOR_CURR_MAX = 52.6
  MOTOR_WIND_CROSS_SECT = 2.01
  MOTOR_STATOR_RESISTANCE = 0.62
  MOTOR_STATOR_INDUCTANCE = 0.00721
  MOTOR_INERTIA = 0.00148
  MOTOR_COMMUT_OFFSET = 1000000
  MOTOR_WIND_TEMP_MAX = 110
  MOTOR_TAU_THERM = 2760
  MOTOR_AMB_TEMP_RATED = 40
  MOTOR_TEMPMODEL_REFSENS = 0
  MOTOR_TEMPMODEL_RES1 = 0
  MOTOR_TEMPMODEL_CAP1 = 0
  MOTOR_TEMPMODEL_RES2 = 0
  MOTOR_TEMPMODEL_CAP2 = 0
  MOTOR_TEMPMODEL_LOSS1 = 0
  MOTOR_TEMPMODEL_LOSS2 = 0
  MOTOR_TEMPMODEL_MODE = 16#FFFF
  MOTOR_ENCOD_TEMP_LIM = 120
8LSA75.DB030S000-3 : 8LSA75.DB030S000-3 v1.0.5.34 (Disabled=true)  [EC -> 8AC126.60-1b.EC; MT -> 8V1180.001-2_L_Carriage.MT1]
  MOTOR_TYPE = 16#0002
  MOTOR_COMPATIBILITY = 16#0207
  MOTOR_WIND_CONNECT = 1
  MOTOR_BRAKE_TYPE = 0
  MOTOR_BRAKE_CURR_RATED = 0
  MOTOR_BRAKE_TORQ_RATED = 0
  MOTOR_BRAKE_ON_TIME = 0
  MOTOR_BRAKE_OFF_TIME = 0
  MOTOR_BRAKE_RESISTANCE = 0
  MOTOR_BRAKE_INDUCTANCE = 0
  MOTOR_BRAKE_VOLT_REL = 0
  MOTOR_BRAKE_VOLT_HOLD = 0
  MOTOR_BRAKE_VOLT_MAX = 0
  MOTOR_TEMPSENS_PAR1 = 31
  MOTOR_TEMPSENS_PAR2 = 289
  MOTOR_TEMPSENS_PAR3 = -30
  MOTOR_TEMPSENS_PAR4 = -0.65
  MOTOR_TEMPSENS_PAR5 = 29.06
  MOTOR_TEMPSENS_PAR6 = 58.83
  MOTOR_TEMPSENS_PAR7 = 88.17
  MOTOR_TEMPSENS_PAR8 = 117.42
  MOTOR_TEMPSENS_PAR9 = 147.14
  MOTOR_TEMPSENS_PAR10 = 175
  MOTOR_TEMPSENS_TYPE = 4353
  MOTOR_TEMPSENS_LIM = 130
  MOTOR_POLEPAIRS = 5
  MOTOR_VOLTAGE_RATED = 400
  MOTOR_VOLTAGE_CONST = 98.44
  MOTOR_SPEED_RATED = 3000
  MOTOR_SPEED_MAX = 4500
  MOTOR_TORQ_STALL = 43
  MOTOR_TORQ_RATED = 30
  MOTOR_TORQ_MAX = 187
  MOTOR_TORQ_CONST = 1.63
  MOTOR_CURR_STALL = 26.4
  MOTOR_CURR_RATED = 18.4
  MOTOR_CURR_MAX = 168.71
  MOTOR_WIND_CROSS_SECT = 4.36
  MOTOR_STATOR_RESISTANCE = 0.21
  MOTOR_STATOR_INDUCTANCE = 0.0039
  MOTOR_INERTIA = 0.0074
  MOTOR_COMMUT_OFFSET = 1000000
  MOTOR_WIND_TEMP_MAX = 110
  MOTOR_TAU_THERM = 2760
  MOTOR_AMB_TEMP_RATED = 40
  MOTOR_TEMPMODEL_REFSENS = 0
  MOTOR_TEMPMODEL_RES1 = 0
  MOTOR_TEMPMODEL_CAP1 = 0
  MOTOR_TEMPMODEL_RES2 = 0
  MOTOR_TEMPMODEL_CAP2 = 0
  MOTOR_TEMPMODEL_LOSS1 = 0
  MOTOR_TEMPMODEL_LOSS2 = 0
  MOTOR_TEMPMODEL_MODE = 16#FFFF
  MOTOR_ENCOD_TEMP_LIM = 120
8LSA75.DB030S000-3a : 8LSA75.DB030S000-3 v1.0.5.34 (Disabled=true)  [EC -> 8AC126.60-1c.EC; MT -> 8V1180.001-2a_R_Carriage.MT1]
  MOTOR_TYPE = 16#0002
  MOTOR_COMPATIBILITY = 16#0207
  MOTOR_WIND_CONNECT = 1
  MOTOR_BRAKE_TYPE = 0
  MOTOR_BRAKE_CURR_RATED = 0
  MOTOR_BRAKE_TORQ_RATED = 0
  MOTOR_BRAKE_ON_TIME = 0
  MOTOR_BRAKE_OFF_TIME = 0
  MOTOR_BRAKE_RESISTANCE = 0
  MOTOR_BRAKE_INDUCTANCE = 0
  MOTOR_BRAKE_VOLT_REL = 0
  MOTOR_BRAKE_VOLT_HOLD = 0
  MOTOR_BRAKE_VOLT_MAX = 0
  MOTOR_TEMPSENS_PAR1 = 31
  MOTOR_TEMPSENS_PAR2 = 289
  MOTOR_TEMPSENS_PAR3 = -30
  MOTOR_TEMPSENS_PAR4 = -0.65
  MOTOR_TEMPSENS_PAR5 = 29.06
  MOTOR_TEMPSENS_PAR6 = 58.83
  MOTOR_TEMPSENS_PAR7 = 88.17
  MOTOR_TEMPSENS_PAR8 = 117.42
  MOTOR_TEMPSENS_PAR9 = 147.14
  MOTOR_TEMPSENS_PAR10 = 175
  MOTOR_TEMPSENS_TYPE = 4353
  MOTOR_TEMPSENS_LIM = 130
  MOTOR_POLEPAIRS = 5
  MOTOR_VOLTAGE_RATED = 400
  MOTOR_VOLTAGE_CONST = 98.44
  MOTOR_SPEED_RATED = 3000
  MOTOR_SPEED_MAX = 4500
  MOTOR_TORQ_STALL = 43
  MOTOR_TORQ_RATED = 30
  MOTOR_TORQ_MAX = 187
  MOTOR_TORQ_CONST = 1.63
  MOTOR_CURR_STALL = 26.4
  MOTOR_CURR_RATED = 18.4
  MOTOR_CURR_MAX = 168.71
  MOTOR_WIND_CROSS_SECT = 4.36
  MOTOR_STATOR_RESISTANCE = 0.21
  MOTOR_STATOR_INDUCTANCE = 0.0039
  MOTOR_INERTIA = 0.0074
  MOTOR_COMMUT_OFFSET = 1000000
  MOTOR_WIND_TEMP_MAX = 110
  MOTOR_TAU_THERM = 2760
  MOTOR_AMB_TEMP_RATED = 40
  MOTOR_TEMPMODEL_REFSENS = 0
  MOTOR_TEMPMODEL_RES1 = 0
  MOTOR_TEMPMODEL_CAP1 = 0
  MOTOR_TEMPMODEL_RES2 = 0
  MOTOR_TEMPMODEL_CAP2 = 0
  MOTOR_TEMPMODEL_LOSS1 = 0
  MOTOR_TEMPMODEL_LOSS2 = 0
  MOTOR_TEMPMODEL_MODE = 16#FFFF
  MOTOR_ENCOD_TEMP_LIM = 120
8V1090.001-2_L_BlowPin : 8V1090.001-2 v1.0.0.0 (Disabled=true)  // Left Blow Pin ACOPOS servo drive, 3x 400-480 V, 8.8 A, 4 kW, coated, line filter, braking resistor and electronic...
8V1090.001-2a_R_BlowPin : 8V1090.001-2 v1.0.0.0 (Disabled=true)
8V1180.001-2_L_Carriage : 8V1180.001-2 v1.0.0.0 (Disabled=true)
8V1180.001-2a_R_Carriage : 8V1180.001-2 v1.0.0.0 (Disabled=true)
FEPL-02_and_ACS580 : FBE.000000B7_ACS580_v2.06.0.0_FEPL-02_1.0 v1.0.0.0 (OrderNumber=FEPL-02 and ACS580)  [PLK1 -> X20BC0083.PLK2 (NodeNumber=20); PLK2 -> FEPL-02_and_ACS580a.PLK1 (NodeNumber=20)]
  Supervision = off
  p2101_direction = wo
  p2102_direction = wo
  p2103_direction = wo
  p2104_direction = ro
  p2105_direction = ro
  p2106_direction = ro
  p603F_direction = ro
  p4001s06_direction = ro
  p4001s07_direction = ro
  p4001s0B_direction = ro
  p4001s0E_direction = ro
FEPL-02_and_ACS580a : FBE.000000B7_ACS580_v2.06.0.0_FEPL-02_1.0 v1.0.0.0 (OrderNumber=FEPL-02 and ACS580)  [PLK1 -> FEPL-02_and_ACS580.PLK2 (NodeNumber=23); PLK2 -> FEPL-02_and_ACS580a1.PLK1 (NodeNumber=23)]
  Supervision = off
  p2101_direction = wo
  p2102_direction = wo
  p2103_direction = wo
  p2104_direction = ro
  p2105_direction = ro
  p2106_direction = ro
  p603F_direction = ro
  p4001s06_direction = ro
  p4001s07_direction = ro
  p4001s0B_direction = ro
  p4001s0E_direction = ro
FEPL-02_and_ACS580a1 : FBE.000000B7_ACS580_v2.06.0.0_FEPL-02_1.0 v1.0.0.0 (OrderNumber=FEPL-02 and ACS580)  [PLK1 -> FEPL-02_and_ACS580a.PLK2 (NodeNumber=24)]
  Supervision = off
  p2101_direction = wo
  p2102_direction = wo
  p2103_direction = wo
  p2104_direction = ro
  p2105_direction = ro
  p2106_direction = ro
  p603F_direction = ro
  p4001s06_direction = ro
  p4001s07_direction = ro
  p4001s0B_direction = ro
  p4001s0E_direction = ro
FEPL-02_and_ACS580a2 : FBE.000000B7_ACS580_v2.06.0.0_FEPL-02_1.0 v1.0.0.0 (Disabled=true, OrderNumber=FEPL-02 and ACS580)
  Supervision = off
  p2101_direction = wo
  p2102_direction = wo
  p2103_direction = wo
  p2104_direction = ro
  p2105_direction = ro
  p2106_direction = ro
  p603F_direction = ro
  p4001s06_direction = ro
  p4001s07_direction = ro
  p4001s0B_direction = ro
  p4001s0E_direction = ro
FEPL-02_and_ACS580a2a : FBE.000000B7_ACS580_v2.06.0.0_FEPL-02_1.0 v1.0.0.0 (Disabled=true, OrderNumber=FEPL-02 and ACS580)
  Supervision = off
  p2101_direction = wo
  p2102_direction = wo
  p2103_direction = wo
  p2104_direction = ro
  p2105_direction = ro
  p2106_direction = ro
  p603F_direction = ro
  p4001s06_direction = ro
  p4001s07_direction = ro
  p4001s0B_direction = ro
  p4001s0E_direction = ro
L-Carriage : MotorSynchronous_any v1.0.1.0  [EC -> 8BAC0120.001-2b.EC; MT -> 8BVI0330HWS0.000-1a.MT1]
  MOTOR_POLEPAIRS = 7
  BrakeAvailable = False
  TempSensType = PTCSwitch
  MOTOR_TEMPSENS_PAR1 = 550
  MOTOR_TEMPSENS_PAR2 = 100
  MOTOR_TEMPSENS_PAR3 = 140
  MOTOR_VOLTAGE_RATED = 400
  MOTOR_VOLTAGE_CONST = 99
  MOTOR_SPEED_RATED = 4500
  MOTOR_SPEED_MAX = 4500
  MOTOR_TORQ_STALL = 20.0
  MOTOR_TORQ_RATED = 12.1
  MOTOR_TORQ_MAX = 65
  MOTOR_TORQ_CONST = 1.052174
  MOTOR_CURR_STALL = 17.8
  MOTOR_CURR_RATED = 11.5
  MOTOR_CURR_MAX = 78
  MOTOR_WIND_CROSS_SECT = 0
  MOTOR_STATOR_RESISTANCE = 0.54246038
  MOTOR_STATOR_INDUCTANCE = 0.0036084116
  MOTOR_INERTIA = 0.0021599999
  MOTOR_COMMUT_OFFSET = 0.044620514
  MOTOR_TAU_THERM = 3000
  MOTOR_WIND_TEMP_MAX = 100
L-Clamp : MotorSynchronous_any v1.0.1.0 (Disabled=true)  [EC -> 8BAC0120.001-2g.EC; MT -> 8BVI0440HWS0.000-1a.MT1]
  MOTOR_POLEPAIRS = 8
  BrakeAvailable = False
  TempSensType = PTCSwitch
  MOTOR_TEMPSENS_PAR1 = 550
  MOTOR_TEMPSENS_PAR2 = 100
  MOTOR_TEMPSENS_PAR3 = 140
  MOTOR_VOLTAGE_RATED = 400
  MOTOR_VOLTAGE_CONST = 136
  MOTOR_SPEED_RATED = 3000
  MOTOR_SPEED_MAX = 3000
  MOTOR_TORQ_STALL = 37.1
  MOTOR_TORQ_RATED = 22.3
  MOTOR_TORQ_MAX = 100
  MOTOR_TORQ_CONST = 1.68
  MOTOR_CURR_STALL = 22.3
  MOTOR_CURR_RATED = 13.9
  MOTOR_CURR_MAX = 84
  MOTOR_WIND_CROSS_SECT = 0
  MOTOR_STATOR_RESISTANCE = 0.3
  MOTOR_STATOR_INDUCTANCE = 0.005
  MOTOR_INERTIA = 0.0058
  MOTOR_COMMUT_OFFSET = 0.044620514
  MOTOR_TAU_THERM = 3000
  MOTOR_WIND_TEMP_MAX = 100
R-BlowPin : MotorSynchronous_any v1.0.1.0  [EC -> 8BAC0120.001-2d.EC; MT -> 8BVI0110HWD0.000-1.MT2]
  MOTOR_POLEPAIRS = 7
  MOTOR_BRAKE_CURR_RATED = 1
  MOTOR_BRAKE_TORQ_RATED = 12
  MOTOR_BRAKE_ON_TIME = 0.01
  MOTOR_BRAKE_OFF_TIME = 0.1
  TempSensType = PTCSwitch
  MOTOR_TEMPSENS_PAR1 = 550
  MOTOR_TEMPSENS_PAR2 = 100
  MOTOR_TEMPSENS_PAR3 = 140
  MOTOR_VOLTAGE_RATED = 400
  MOTOR_VOLTAGE_CONST = 75.673531
  MOTOR_SPEED_RATED = 3000
  MOTOR_SPEED_MAX = 6000
  MOTOR_TORQ_STALL = 9.6000004
  MOTOR_TORQ_RATED = 9.6000004
  MOTOR_TORQ_MAX = 43
  MOTOR_TORQ_CONST = 1.2516297
  MOTOR_CURR_STALL = 7.6700001
  MOTOR_CURR_RATED = 7.67
  MOTOR_CURR_MAX = 41
  MOTOR_WIND_CROSS_SECT = 0
  MOTOR_STATOR_RESISTANCE = 1.6416402
  MOTOR_STATOR_INDUCTANCE = 0.0092184199
  MOTOR_INERTIA = 0.00075800001
  MOTOR_COMMUT_OFFSET = -0.003623
  MOTOR_TAU_THERM = 3000
  MOTOR_WIND_TEMP_MAX = 100
R-Carriage : MotorSynchronous_any v1.0.1.0 (Disabled=true)  [EC -> 8BAC0120.001-2.EC; MT -> 8BVI0330HWS0.000-1.MT1]
  MOTOR_POLEPAIRS = 7
  BrakeAvailable = False
  TempSensType = PTCSwitch
  MOTOR_TEMPSENS_PAR1 = 550
  MOTOR_TEMPSENS_PAR2 = 100
  MOTOR_TEMPSENS_PAR3 = 140
  MOTOR_VOLTAGE_RATED = 400
  MOTOR_VOLTAGE_CONST = 63.614437
  MOTOR_SPEED_RATED = 4500
  MOTOR_SPEED_MAX = 4500
  MOTOR_TORQ_STALL = 12.1
  MOTOR_TORQ_RATED = 12.1
  MOTOR_TORQ_MAX = 65
  MOTOR_TORQ_CONST = 1.052174
  MOTOR_CURR_STALL = 11.5
  MOTOR_CURR_RATED = 11.5
  MOTOR_CURR_MAX = 78
  MOTOR_WIND_CROSS_SECT = 0
  MOTOR_STATOR_RESISTANCE = 0.53999424
  MOTOR_STATOR_INDUCTANCE = 0.003565806
  MOTOR_INERTIA = 0.0021599999
  MOTOR_COMMUT_OFFSET = 0.091310501
  MOTOR_TAU_THERM = 3000
  MOTOR_WIND_TEMP_MAX = 100
R-Clamp : MotorSynchronous_any v1.0.1.0
  MOTOR_POLEPAIRS = 8
  BrakeAvailable = False
  TempSensType = PTCSwitch
  MOTOR_TEMPSENS_PAR1 = 550
  MOTOR_TEMPSENS_PAR2 = 100
  MOTOR_TEMPSENS_PAR3 = 140
  MOTOR_VOLTAGE_RATED = 400
  MOTOR_VOLTAGE_CONST = 96.996979
  MOTOR_SPEED_RATED = 3000
  MOTOR_SPEED_MAX = 3000
  MOTOR_TORQ_STALL = 22.3
  MOTOR_TORQ_RATED = 22.3
  MOTOR_TORQ_MAX = 100
  MOTOR_TORQ_CONST = 1.6043166
  MOTOR_CURR_STALL = 13.9
  MOTOR_CURR_RATED = 13.9
  MOTOR_CURR_MAX = 84
  MOTOR_WIND_CROSS_SECT = 0
  MOTOR_STATOR_RESISTANCE = 0.40099636
  MOTOR_STATOR_INDUCTANCE = 0.003689728
  MOTOR_INERTIA = 0.0058
  MOTOR_COMMUT_OFFSET = 0.026538849
  MOTOR_TAU_THERM = 3000
  MOTOR_WIND_TEMP_MAX = 100
R-Clamp1 : MotorSynchronous_any v1.0.1.0 (Disabled=true)  [EC -> 8BAC0120.001-2i.EC; MT -> 8BVI0440HWS0.000-1.MT1]
  MOTOR_POLEPAIRS = 8
  BrakeAvailable = False
  TempSensType = PTCSwitch
  MOTOR_TEMPSENS_PAR1 = 550
  MOTOR_TEMPSENS_PAR2 = 100
  MOTOR_TEMPSENS_PAR3 = 140
  MOTOR_VOLTAGE_RATED = 400
  MOTOR_VOLTAGE_CONST = 112
  MOTOR_SPEED_RATED = 2000
  MOTOR_SPEED_MAX = 4000
  MOTOR_TORQ_STALL = 66.1
  MOTOR_TORQ_RATED = 43.7
  MOTOR_TORQ_MAX = 205
  MOTOR_TORQ_CONST = 1.75
  MOTOR_CURR_STALL = 37.9
  MOTOR_CURR_RATED = 25.9
  MOTOR_CURR_MAX = 155
  MOTOR_WIND_CROSS_SECT = 0
  MOTOR_STATOR_RESISTANCE = 0.13
  MOTOR_STATOR_INDUCTANCE = 0.00222
  MOTOR_INERTIA = 0.0133
  MOTOR_COMMUT_OFFSET = -0.031101227
  MOTOR_TAU_THERM = 3000
  MOTOR_WIND_TEMP_MAX = 100
Thick : MotorSynchronous_any v1.0.1.0  [EC -> 8BAC0120.001-2c.EC; MT -> 8BVI0110HWD0.000-1.MT1]
  MOTOR_POLEPAIRS = 7
  MOTOR_BRAKE_CURR_RATED = 1.1
  MOTOR_BRAKE_TORQ_RATED = 32
  MOTOR_BRAKE_ON_TIME = 0.02
  MOTOR_BRAKE_OFF_TIME = 0.01
  TempSensType = PTCSwitch
  MOTOR_TEMPSENS_PAR1 = 550
  MOTOR_TEMPSENS_PAR2 = 100
  MOTOR_TEMPSENS_PAR3 = 140
  MOTOR_VOLTAGE_RATED = 400
  MOTOR_VOLTAGE_CONST = 87.507896
  MOTOR_SPEED_RATED = 3000
  MOTOR_SPEED_MAX = 3000
  MOTOR_TORQ_STALL = 16.5
  MOTOR_TORQ_RATED = 16.5
  MOTOR_TORQ_MAX = 65
  MOTOR_TORQ_CONST = 1.4473685
  MOTOR_CURR_STALL = 11.4
  MOTOR_CURR_RATED = 11.4
  MOTOR_CURR_MAX = 62
  MOTOR_WIND_CROSS_SECT = 0
  MOTOR_STATOR_RESISTANCE = 0.80327398
  MOTOR_STATOR_INDUCTANCE = 0.0053170878
  MOTOR_INERTIA = 0.00216
  MOTOR_COMMUT_OFFSET = -0.01932621
  MOTOR_TAU_THERM = 3000
  MOTOR_WIND_TEMP_MAX = 100
X20AI4632_A : X20AI4632 v1.2.0.0  [SS1 -> X20TB12g.SS; SL -> X20BM11k.SL1]
  Supervision = off
X20AI4632_B : X20AI4632 v1.2.0.0  [SS1 -> X20TB12h.SS; SL -> X20BM11l.SL1]
  Supervision = off
X20AI4632_C : X20AI4632 v1.2.0.0 (Disabled=true)  [SS1 -> X20TB12p.SS; SL -> X20BM11ac.SL1]
  Supervision = off
  ChannelType01 = 0 to 20mA
  ChannelType02 = 0 to 20mA
  ChannelType03 = 0 to 20mA
  ChannelType04 = 0 to 20mA
X20AO4622_A : X20AO4622 v1.2.0.0 (Disabled=true)  [SS1 -> X20TB12i.SS; SL -> X20BM11m.SL1]
  Supervision = off
X20AO4622_B : X20AO4622 v1.2.0.0 (Disabled=true)  [SS1 -> X20TB12j.SS; SL -> X20BM11n.SL1]
  Supervision = off
X20AO4632_A : X20AO4632 v1.1.0.0  [SS1 -> X20TB12r.SS; SL -> X20BM11ad.SL1]
  Supervision = off
X20AO4632_B : X20AO4632 v1.1.0.0  [SS1 -> X20TB12s.SS; SL -> X20BM11ae.SL1]
  Supervision = off
X20AO4632_C : X20AO4632 v1.1.0.0 (Disabled=true)  [SS1 -> X20TB12t.SS; SL -> X20BM11af.SL1]
  Supervision = off
X20AO4632_D : X20AO4632 v1.1.0.0 (Disabled=true)  [SS1 -> X20TB12u.SS; SL -> X20BM11ag.SL1]
  Supervision = off
X20AP3131_A : X20AP3131 v1.4.0.0 (Disabled=true)  [SS1 -> X20TB32.SS; SL -> X20BM32.SL1]
  Supervision = off
  EnergyUnit = 1Wh
  DisIrmsA = on
  DisIrmsB = on
  DisIrmsC = on
  DisQmeanT = off
  DisReacEnT = off
X20AP3131_B : X20AP3131 v1.4.0.0 (Disabled=true)  [SS1 -> X20TB32a.SS; SL -> X20BM32a.SL1]
  Supervision = off
  EnergyUnit = 1Wh
  DisIrmsA = on
  DisIrmsB = on
  DisIrmsC = on
  DisQmeanT = off
  DisReacEnT = off
X20AP3131_C : X20AP3131 v1.4.0.0 (Disabled=true)  [SS1 -> X20TB32b.SS; SL -> X20BM32b.SL1]
  Supervision = off
  EnergyUnit = 1Wh
  DisIrmsA = on
  DisIrmsB = on
  DisIrmsC = on
  DisQmeanT = off
  DisReacEnT = off
X20ATC402_A : X20ATC402 v1.0.2.0  [SS1 -> X20TB1E.SS; SL -> X20BM11q.SL1]
  Supervision = off
  InputFilter = 66.7ms
  Temp01 = on
  SensorType01 = Typ_K
  Ref01 = Reference_B
  Temp02 = on
  SensorType02 = Typ_K
  Ref02 = Reference_B
  Temp03 = on
  SensorType03 = Typ_K
  Ref03 = Reference_B
  Temp04 = on
  SensorType04 = Typ_K
  Ref04 = Reference_B
  Temp05 = on
  SensorType05 = Typ_K
  Ref05 = Reference_B
  Temp06 = on
  SensorType06 = Typ_K
  Ref06 = Reference_B
X20ATC402_B : X20ATC402 v1.0.2.0  [SS1 -> X20TB1E1.SS; SL -> X20BM11r.SL1]
  Supervision = off
  InputFilter = 66.7ms
  Temp01 = on
  SensorType01 = Typ_K
  Ref01 = Reference_B
  Temp02 = on
  SensorType02 = Typ_K
  Ref02 = Reference_B
  Temp03 = on
  SensorType03 = Typ_K
  Ref03 = Reference_B
  Temp04 = on
  SensorType04 = Typ_K
  Ref04 = Reference_B
  Temp05 = on
  SensorType05 = Typ_K
  Ref05 = Reference_B
  Temp06 = on
  SensorType06 = Typ_K
  Ref06 = Reference_B
X20ATC402_C : X20ATC402 v1.0.2.0  [SS1 -> X20TB1E2.SS; SL -> X20BM11s.SL1]
  Supervision = off
  InputFilter = 66.7ms
  Temp01 = on
  SensorType01 = Typ_K
  Ref01 = Reference_B
  Temp02 = on
  SensorType02 = Typ_K
  Ref02 = Reference_B
  Temp03 = on
  SensorType03 = Typ_K
  Ref03 = Reference_B
  Temp04 = on
  SensorType04 = Typ_K
  Ref04 = Reference_B
  Temp05 = on
  SensorType05 = Typ_K
  Ref05 = Reference_B
  Temp06 = on
  SensorType06 = Typ_K
  Ref06 = Reference_B
X20ATC402_D : X20ATC402 v1.0.2.0 (Disabled=true)  [SS1 -> X20TB1E3.SS; SL -> X20BM11t.SL1]
  Supervision = off
  InputFilter = 66.7ms
  Temp01 = on
  SensorType01 = Typ_K
  Ref01 = Reference_B
  Temp02 = on
  SensorType02 = Typ_K
  Ref02 = Reference_B
  Temp03 = on
  SensorType03 = Typ_K
  Ref03 = Reference_B
  Temp04 = on
  SensorType04 = Typ_K
  Ref04 = Reference_B
  Temp05 = on
  SensorType05 = Typ_K
  Ref05 = Reference_B
  Temp06 = on
  SensorType06 = Typ_K
  Ref06 = Reference_B
X20ATC402_E : X20ATC402 v1.0.2.0 (Disabled=true)  [SS1 -> X20TB1E4.SS; SL -> X20BM11u.SL1]
  Supervision = off
  InputFilter = 66.7ms
  Temp01 = on
  SensorType01 = Typ_K
  Ref01 = Reference_B
  Temp02 = on
  SensorType02 = Typ_K
  Ref02 = Reference_B
  Temp03 = on
  SensorType03 = Typ_K
  Ref03 = Reference_B
  Temp04 = on
  SensorType04 = Typ_K
  Ref04 = Reference_B
  Temp05 = on
  SensorType05 = Typ_K
  Ref05 = Reference_B
  Temp06 = on
  SensorType06 = Typ_K
  Ref06 = Reference_B
X20ATC402_F : X20ATC402 v1.0.2.0 (Disabled=true)  [SS1 -> X20TB1E5.SS; SL -> X20BM11ab.SL1]
  Supervision = off
  InputFilter = 66.7ms
  Temp01 = on
  SensorType01 = Typ_K
  Ref01 = Reference_B
  Temp02 = on
  SensorType02 = Typ_K
  Ref02 = Reference_B
  Temp03 = on
  SensorType03 = Typ_K
  Ref03 = Reference_B
  Temp04 = on
  SensorType04 = Typ_K
  Ref04 = Reference_B
  Temp05 = on
  SensorType05 = Typ_K
  Ref05 = Reference_B
  Temp06 = on
  SensorType06 = Typ_K
  Ref06 = Reference_B
X20BB80 : X20BB80 v1.0.2.0
X20BB80a : X20BB80 v1.0.2.0 (Disabled=true)
  Connector IF1 (Disabled=true)
X20BB80b : X20BB80 v1.0.2.0 (Disabled=true)
  Connector IF1 (Disabled=true)
X20BC0083 : X20BC0083 v2.9.0.0  [PLK1 -> 5ACCIF01.FPSC-001.IF1 (NodeNumber=2); PLK2 -> FEPL-02_and_ACS580.PLK1 (NodeNumber=2); SL -> X20BB80.SL1]
  Supervision = off
X20BC0083a : X20BC0083 v2.9.0.0 (Disabled=true)  [PLK2 -> 8AC114.60-2.PLK1 (NodeNumber=2); SL -> X20BB80a.SL1]
  Supervision = off
X20BC0083b : X20BC0083 v2.9.0.0 (Disabled=true)  [SL -> X20BB80b.SL1]
  Supervision = off
X20BM01 : X20BM01 v2.1.0.0  [X2X1 -> X20BM11g.X2X2]
X20BM01a : X20BM01 v2.1.0.0 (Disabled=true)  [X2X1 -> X20BM11y.X2X2]
X20BM11 : X20BM11 v1.0.0.1  [X2X1 -> X20BB80.IF1]
X20BM11a : X20BM11 v1.0.0.1  [X2X1 -> X20BM11.X2X2]
X20BM11aa : X20BM11 v1.0.0.1 (Disabled=true)  [X2X1 -> X20BM11ag.X2X2]
X20BM11ab : X20BM11 v1.0.0.1 (Disabled=true)  [X2X1 -> X20BM11u.X2X2]
X20BM11ac : X20BM11 v1.0.0.1 (Disabled=true)  [X2X1 -> X20BM11s.X2X2]
X20BM11ad : X20BM11 v1.0.0.1  [X2X1 -> X20BM11l.X2X2]
X20BM11ae : X20BM11 v1.0.0.1  [X2X1 -> X20BM11ad.X2X2]
X20BM11af : X20BM11 v1.0.0.1 (Disabled=true)  [X2X1 -> X20BM11ac.X2X2]
X20BM11ag : X20BM11 v1.0.0.1 (Disabled=true)  [X2X1 -> X20BM11af.X2X2]
X20BM11b : X20BM11 v1.0.0.1  [X2X1 -> X20BM11a.X2X2]
X20BM11c : X20BM11 v1.0.0.1  [X2X1 -> X20BM11b.X2X2]
X20BM11d : X20BM11 v1.0.0.1  [X2X1 -> X20BM11c.X2X2]
X20BM11e : X20BM11 v1.0.0.1  [X2X1 -> X20BM11d.X2X2]
X20BM11f : X20BM11 v1.0.0.1  [X2X1 -> X20BM11e.X2X2]
X20BM11g : X20BM11 v1.0.0.1  [X2X1 -> X20BM11f.X2X2]
X20BM11h : X20BM11 v1.0.0.1  [X2X1 -> X20BM01.X2X2]
X20BM11i : X20BM11 v1.0.0.1  [X2X1 -> X20BM11h.X2X2]
X20BM11j : X20BM11 v1.0.0.1 (Disabled=true)  [X2X1 -> X20BB80b.IF1]
X20BM11k : X20BM11 v1.0.0.1  [X2X1 -> X20BM11i.X2X2]
X20BM11l : X20BM11 v1.0.0.1  [X2X1 -> X20BM11k.X2X2]
X20BM11m : X20BM11 v1.0.0.1 (Disabled=true)  [X2X1 -> X20BM01a.X2X2]
X20BM11n : X20BM11 v1.0.0.1 (Disabled=true)  [X2X1 -> X20BM11m.X2X2]
X20BM11o : X20BM11 v1.0.0.1 (Disabled=true)  [X2X1 -> X20BM11n.X2X2]
X20BM11p : X20BM11 v1.0.0.1 (Disabled=true)  [X2X1 -> X20BM11j.X2X2]
X20BM11q : X20BM11 v1.0.0.1  [X2X1 -> X20BM11ae.X2X2]
X20BM11r : X20BM11 v1.0.0.1  [X2X1 -> X20BM11q.X2X2]
X20BM11s : X20BM11 v1.0.0.1  [X2X1 -> X20BM11r.X2X2]
X20BM11t : X20BM11 v1.0.0.1 (Disabled=true)  [X2X1 -> X20BM11z.X2X2]
X20BM11u : X20BM11 v1.0.0.1 (Disabled=true)  [X2X1 -> X20BM11t.X2X2]
X20BM11v : X20BM11 v1.0.0.1 (Disabled=true)  [X2X1 -> X20BM11aa.X2X2]
X20BM11w : X20BM11 v1.0.0.1 (Disabled=true)  [X2X1 -> X20BM11v.X2X2]
X20BM11x : X20BM11 v1.0.0.1 (Disabled=true)  [X2X1 -> X20BM11w.X2X2]
X20BM11y : X20BM11 v1.0.0.1 (Disabled=true)  [X2X1 -> X20BM11x.X2X2]
X20BM11z : X20BM11 v1.0.0.1 (Disabled=true)  [X2X1 -> X20BM11p.X2X2]
X20BM32 : X20BM32 v1.0.0.1 (Disabled=true)  [X2X1 -> X20BM11o.X2X2]
X20BM32a : X20BM32 v1.0.0.1 (Disabled=true)  [X2X1 -> X20BM32.X2X2]
X20BM32b : X20BM32 v1.0.0.1 (Disabled=true)  [X2X1 -> X20BM32a.X2X2]
X20DIF371_A : X20DIF371 v1.0.1.0  [SS1 -> X20TB1F.SS; SL -> X20BM11.SL1]
  Supervision = off
X20DIF371_B : X20DIF371 v1.0.1.0  [SS1 -> X20TB1F1.SS; SL -> X20BM11a.SL1]
  Supervision = off
X20DIF371_C : X20DIF371 v1.0.1.0  [SS1 -> X20TB1F2.SS; SL -> X20BM11b.SL1]
  Supervision = off
X20DIF371_D : X20DIF371 v1.0.1.0 (Disabled=true)  [SS1 -> X20TB1F9.SS; SL -> X20BM11aa.SL1]
  Supervision = off
X20DO8332_A : X20DO8332 v1.3.0.0  [SS1 -> X20TB12b.SS; SL -> X20BM11c.SL1]
  Supervision = off
X20DO8332_B : X20DO8332 v1.3.0.0  [SS1 -> X20TB12c.SS; SL -> X20BM11d.SL1]
  Supervision = off
X20DO8332_C : X20DO8332 v1.3.0.0  [SS1 -> X20TB12d.SS; SL -> X20BM11e.SL1]
  Supervision = off
X20DO8332_D : X20DO8332 v1.3.0.0  [SS1 -> X20TB12e.SS; SL -> X20BM11f.SL1]
  Supervision = off
X20DO8332_E : X20DO8332 v1.3.0.0 (Disabled=true)  [SS1 -> X20TB12l.SS; SL -> X20BM11v.SL1]
  Supervision = off
X20DO8332_F : X20DO8332 v1.3.0.0 (Disabled=true)  [SS1 -> X20TB12m.SS; SL -> X20BM11w.SL1]
  Supervision = off
X20DO8332_G : X20DO8332 v1.3.0.0 (Disabled=true)  [SS1 -> X20TB12n.SS; SL -> X20BM11x.SL1]
  Supervision = off
X20DO8332_H : X20DO8332 v1.3.0.0 (Disabled=true)  [SS1 -> X20TB12o.SS; SL -> X20BM11y.SL1]
  Supervision = off
X20DOF322_A : X20DOF322 v1.4.0.0  [SS1 -> X20TB1F3.SS; SL -> X20BM11g.SL1]
  Supervision = off
X20DOF322_B : X20DOF322 v1.4.0.0  [SS1 -> X20TB1F4.SS; SL -> X20BM11h.SL1]
  Supervision = off
X20DOF322_C : X20DOF322 v1.4.0.0  [SS1 -> X20TB1F5.SS; SL -> X20BM11i.SL1]
  Supervision = off
X20DOF322_D : X20DOF322 v1.4.0.0 (Disabled=true)  [SS1 -> X20TB1F6.SS; SL -> X20BM11j.SL1]
  Supervision = off
X20DOF322_E : X20DOF322 v1.4.0.0 (Disabled=true)  [SS1 -> X20TB1F7.SS; SL -> X20BM11p.SL1]
  Supervision = off
X20DOF322_F : X20DOF322 v1.4.0.0 (Disabled=true)  [SS1 -> X20TB1F8.SS; SL -> X20BM11z.SL1]
  Supervision = off
X20DS1119 : X20DS1119 v1.4.1.0 (Disabled=true)  [SS1 -> X20TB12k.SS; SL -> X20BM11o.SL1]
  Supervision = off
  Function03 = AB
X20PS3300 : X20PS3300 v1.1.0.0  [SS1 -> X20TB12f.SS; SL -> X20BM01.SL1]
  Supervision = off
X20PS3300a : X20PS3300 v1.1.0.0 (Disabled=true)  [SS1 -> X20TB12q.SS; SL -> X20BM01a.SL1]
  Supervision = off
X20PS9400 : X20PS9400 v1.0.2.4  [SS1 -> X20TB12.SS; PS -> X20BB80.PS1]
  Supervision = off
X20PS9400a : X20PS9400 v1.0.2.4 (Disabled=true)  [SS1 -> X20TB12a.SS; PS -> X20BB80a.PS1]
  Supervision = off
X20PS9400b : X20PS9400 v1.0.2.4 (Disabled=true)  [SS1 -> X20TB12v.SS; PS -> X20BB80b.PS1]
  Supervision = off
X20TB12 : X20TB12 v1.0.0.0
X20TB12a : X20TB12 v1.0.0.0 (Disabled=true)
X20TB12b : X20TB12 v1.0.0.0
X20TB12c : X20TB12 v1.0.0.0
X20TB12d : X20TB12 v1.0.0.0
X20TB12e : X20TB12 v1.0.0.0
X20TB12f : X20TB12 v1.0.0.0
X20TB12g : X20TB12 v1.0.0.0
X20TB12h : X20TB12 v1.0.0.0
X20TB12i : X20TB12 v1.0.0.0 (Disabled=true)
X20TB12j : X20TB12 v1.0.0.0 (Disabled=true)
X20TB12k : X20TB12 v1.0.0.0 (Disabled=true)
X20TB12l : X20TB12 v1.0.0.0 (Disabled=true)
X20TB12m : X20TB12 v1.0.0.0 (Disabled=true)
X20TB12n : X20TB12 v1.0.0.0 (Disabled=true)
X20TB12o : X20TB12 v1.0.0.0 (Disabled=true)
X20TB12p : X20TB12 v1.0.0.0 (Disabled=true)
X20TB12q : X20TB12 v1.0.0.0 (Disabled=true)
X20TB12r : X20TB12 v1.0.0.0
X20TB12s : X20TB12 v1.0.0.0
X20TB12t : X20TB12 v1.0.0.0 (Disabled=true)
X20TB12u : X20TB12 v1.0.0.0 (Disabled=true)
X20TB12v : X20TB12 v1.0.0.0 (Disabled=true)
X20TB1E : X20TB1E v1.0.0.0
X20TB1E1 : X20TB1E v1.0.0.0
X20TB1E2 : X20TB1E v1.0.0.0
X20TB1E3 : X20TB1E v1.0.0.0 (Disabled=true)
X20TB1E4 : X20TB1E v1.0.0.0 (Disabled=true)
X20TB1E5 : X20TB1E v1.0.0.0 (Disabled=true)
X20TB1F : X20TB1F v1.0.0.0
X20TB1F1 : X20TB1F v1.0.0.0
X20TB1F2 : X20TB1F v1.0.0.0
X20TB1F3 : X20TB1F v1.0.0.0
X20TB1F4 : X20TB1F v1.0.0.0
X20TB1F5 : X20TB1F v1.0.0.0
X20TB1F6 : X20TB1F v1.0.0.0 (Disabled=true)
X20TB1F7 : X20TB1F v1.0.0.0 (Disabled=true)
X20TB1F8 : X20TB1F v1.0.0.0 (Disabled=true)
X20TB1F9 : X20TB1F v1.0.0.0 (Disabled=true)
X20TB32 : X20TB32 v1.0.0.1 (Disabled=true)
X20TB32a : X20TB32 v1.0.0.1 (Disabled=true)
X20TB32b : X20TB32 v1.0.0.1 (Disabled=true)
```

### Cpu.per - 5PPC2100_BY01_000/Cpu.per
```iecst
VAR_CONFIG
	gCycleTimes AT %MD0; (* *)
	gCycleTimesL AT %MD4; (* *)
	gCycleTimesR AT %MD8; (* *)
	gExtruderA AT %M12; (* *)
	gExtruderB AT %M132; (* *)
	gExtruderC AT %M252; (* *)
	gExtruderD AT %M372; (* *)
	gExtruderVisu AT %M492; (* *)
	gHeatingPlan AT %M612; (* *)
	gH_IO AT %M684; (* *)
	gMachineStopDays AT %MD1464; (* *)
	gMachineWorkDays AT %MD1468; (* *)
	gMachineWorkTime AT %MD1472; (* *)
	gMacOption AT %M1476; (* *)
	gSPC_Current AT %M1544; (* *)
	gThickProf AT %M1616; (* *)
	gT_Par AT %M1788; (* *)
END_VAR
```

### IoMap.iom - 5PPC2100_BY01_000/IoMap.iom
```iecst
VAR_CONFIG
	Cyclic#2.::gHardWare.DIF371_4[0] AT %IX."X20DIF371_D".DigitalInput01;
	Cyclic#2.::gHardWare.DIF371_4[1] AT %IX."X20DIF371_D".DigitalInput02;
	Cyclic#2.::gHardWare.DIF371_4[2] AT %IX."X20DIF371_D".DigitalInput03;
	Cyclic#2.::gHardWare.DIF371_4[3] AT %IX."X20DIF371_D".DigitalInput04;
	Cyclic#2.::gHardWare.DIF371_4[4] AT %IX."X20DIF371_D".DigitalInput05;
	Cyclic#2.::gHardWare.DIF371_4[5] AT %IX."X20DIF371_D".DigitalInput06;
	Cyclic#2.::gHardWare.DIF371_4[6] AT %IX."X20DIF371_D".DigitalInput07;
	Cyclic#2.::gHardWare.DIF371_4[7] AT %IX."X20DIF371_D".DigitalInput08;
	Cyclic#2.::gHardWare.DIF371_4[8] AT %IX."X20DIF371_D".DigitalInput09;
	Cyclic#2.::gHardWare.DIF371_4[9] AT %IX."X20DIF371_D".DigitalInput10;
	Cyclic#2.::gHardWare.DIF371_4[10] AT %IX."X20DIF371_D".DigitalInput11;
	Cyclic#2.::gHardWare.DIF371_4[11] AT %IX."X20DIF371_D".DigitalInput12;
	Cyclic#2.::gHardWare.DIF371_4[12] AT %IX."X20DIF371_D".DigitalInput13;
	Cyclic#2.::gHardWare.DIF371_4[13] AT %IX."X20DIF371_D".DigitalInput14;
	Cyclic#2.::gHardWare.DIF371_4[14] AT %IX."X20DIF371_D".DigitalInput15;
	Cyclic#2.::gHardWare.DIF371_4[15] AT %IX."X20DIF371_D".DigitalInput16;
	::gHardWare.DIF371_2[0] AT %IX."X20DIF371a".DigitalInput01;
	::gHardWare.DIF371_2[1] AT %IX."X20DIF371a".DigitalInput02;
	::gHardWare.DIF371_2[2] AT %IX."X20DIF371a".DigitalInput03;
	::gHardWare.DIF371_2[3] AT %IX."X20DIF371a".DigitalInput04;
	::gHardWare.DIF371_2[4] AT %IX."X20DIF371a".DigitalInput05;
	::gHardWare.DIF371_2[5] AT %IX."X20DIF371a".DigitalInput06;
	::gHardWare.DIF371_2[6] AT %IX."X20DIF371a".DigitalInput07;
	::gHardWare.DIF371_2[7] AT %IX."X20DIF371a".DigitalInput08;
	::gHardWare.DIF371_2[8] AT %IX."X20DIF371a".DigitalInput09;
	::gHardWare.DIF371_2[9] AT %IX."X20DIF371a".DigitalInput10;
	::gHardWare.DIF371_2[10] AT %IX."X20DIF371a".DigitalInput11;
	::gHardWare.DIF371_2[11] AT %IX."X20DIF371a".DigitalInput12;
	::gHardWare.DIF371_2[12] AT %IX."X20DIF371a".DigitalInput13;
	::gHardWare.DIF371_2[13] AT %IX."X20DIF371a".DigitalInput14;
	::gHardWare.DIF371_2[14] AT %IX."X20DIF371a".DigitalInput15;
	::gHardWare.DIF371_2[15] AT %IX."X20DIF371a".DigitalInput16;
	Cyclic#2.::gHardWare.DIF371_3[0] AT %IX."X20DIF371_C".DigitalInput01;
	Cyclic#2.::gHardWare.ModuleOk.DIF371_3 AT %IX."X20DIF371_C".ModuleOk;
	Cyclic#2.::gHardWare.DIF371_1[0] AT %IX."X20DIF371_A".DigitalInput01;
	Cyclic#2.::gHardWare.DIF371_1[1] AT %IX."X20DIF371_A".DigitalInput02;
	Cyclic#2.::gHardWare.ModuleOk.DIF371_1 AT %IX."X20DIF371_A".ModuleOk;
	Cyclic#2.::gHardWare.DIF371_1[2] AT %IX."X20DIF371_A".DigitalInput03;
	Cyclic#2.::gHardWare.DIF371_1[3] AT %IX."X20DIF371_A".DigitalInput04;
	Cyclic#2.::gHardWare.DIF371_1[4] AT %IX."X20DIF371_A".DigitalInput05;
	Cyclic#2.::gHardWare.DIF371_1[5] AT %IX."X20DIF371_A".DigitalInput06;
	Cyclic#2.::gHardWare.DIF371_1[6] AT %IX."X20DIF371_A".DigitalInput07;
	Cyclic#2.::gHardWare.DIF371_1[7] AT %IX."X20DIF371_A".DigitalInput08;
	Cyclic#2.::gHardWare.DIF371_1[8] AT %IX."X20DIF371_A".DigitalInput09;
	Cyclic#2.::gHardWare.DIF371_1[9] AT %IX."X20DIF371_A".DigitalInput10;
	Cyclic#2.::gHardWare.DIF371_1[10] AT %IX."X20DIF371_A".DigitalInput11;
	Cyclic#2.::gHardWare.DIF371_1[11] AT %IX."X20DIF371_A".DigitalInput12;
	Cyclic#2.::gHardWare.DIF371_1[12] AT %IX."X20DIF371_A".DigitalInput13;
	Cyclic#2.::gHardWare.DIF371_1[13] AT %IX."X20DIF371_A".DigitalInput14;
	Cyclic#2.::gHardWare.DIF371_1[14] AT %IX."X20DIF371_A".DigitalInput15;
	Cyclic#2.::gHardWare.DIF371_1[15] AT %IX."X20DIF371_A".DigitalInput16;
	Cyclic#2.::gHardWare.DIF371_2[0] AT %IX."X20DIF371_B".DigitalInput01;
	Cyclic#2.::gHardWare.ModuleOk.DIF371_2 AT %IX."X20DIF371_B".ModuleOk;
	Cyclic#2.::gHardWare.DIF371_2[1] AT %IX."X20DIF371_B".DigitalInput02;
	Cyclic#2.::gHardWare.DIF371_2[2] AT %IX."X20DIF371_B".DigitalInput03;
	Cyclic#2.::gHardWare.DIF371_2[3] AT %IX."X20DIF371_B".DigitalInput04;
	Cyclic#2.::gHardWare.DIF371_2[4] AT %IX."X20DIF371_B".DigitalInput05;
	Cyclic#2.::gHardWare.DIF371_2[5] AT %IX."X20DIF371_B".DigitalInput06;
	Cyclic#2.::gHardWare.DIF371_2[6] AT %IX."X20DIF371_B".DigitalInput07;
	Cyclic#2.::gHardWare.DIF371_2[7] AT %IX."X20DIF371_B".DigitalInput08;
	Cyclic#2.::gHardWare.DIF371_2[8] AT %IX."X20DIF371_B".DigitalInput09;
	Cyclic#2.::gHardWare.DIF371_2[9] AT %IX."X20DIF371_B".DigitalInput10;
	Cyclic#2.::gHardWare.DIF371_2[10] AT %IX."X20DIF371_B".DigitalInput11;
	Cyclic#2.::gHardWare.DIF371_2[11] AT %IX."X20DIF371_B".DigitalInput12;
	Cyclic#2.::gHardWare.DIF371_2[12] AT %IX."X20DIF371_B".DigitalInput13;
	Cyclic#2.::gHardWare.DIF371_2[13] AT %IX."X20DIF371_B".DigitalInput14;
	Cyclic#2.::gHardWare.DIF371_2[14] AT %IX."X20DIF371_B".DigitalInput15;
	Cyclic#2.::gHardWare.DIF371_2[15] AT %IX."X20DIF371_B".DigitalInput16;
	Cyclic#2.::gHardWare.DIF371_3[1] AT %IX."X20DIF371_C".DigitalInput02;
	Cyclic#2.::gHardWare.DIF371_3[2] AT %IX."X20DIF371_C".DigitalInput03;
	Cyclic#2.::gHardWare.DIF371_3[3] AT %IX."X20DIF371_C".DigitalInput04;
	Cyclic#2.::gHardWare.DIF371_3[4] AT %IX."X20DIF371_C".DigitalInput05;
	Cyclic#2.::gHardWare.DIF371_3[5] AT %IX."X20DIF371_C".DigitalInput06;
	Cyclic#2.::gHardWare.DIF371_3[6] AT %IX."X20DIF371_C".DigitalInput07;
	Cyclic#2.::gHardWare.DIF371_3[7] AT %IX."X20DIF371_C".DigitalInput08;
	Cyclic#2.::gHardWare.DIF371_3[8] AT %IX."X20DIF371_C".DigitalInput09;
	Cyclic#2.::gHardWare.DIF371_3[9] AT %IX."X20DIF371_C".DigitalInput10;
	Cyclic#2.::gHardWare.DIF371_3[10] AT %IX."X20DIF371_C".DigitalInput11;
	Cyclic#2.::gHardWare.DIF371_3[11] AT %IX."X20DIF371_C".DigitalInput12;
	Cyclic#2.::gHardWare.DIF371_3[12] AT %IX."X20DIF371_C".DigitalInput13;
	Cyclic#2.::gHardWare.DIF371_3[13] AT %IX."X20DIF371_C".DigitalInput14;
	Cyclic#2.::gHardWare.DIF371_3[14] AT %IX."X20DIF371_C".DigitalInput15;
	Cyclic#2.::gHardWare.DIF371_3[15] AT %IX."X20DIF371_C".DigitalInput16;
	Cyclic#2.::gHardWare.ModuleOk.DOF322_1 AT %IX."X20DOF322_A".ModuleOk;
	Cyclic#2.::gHardWare.DOF322_1[0] AT %QX."X20DOF322_A".DigitalOutput01;
	Cyclic#2.::gHardWare.DOF322_1[1] AT %QX."X20DOF322_A".DigitalOutput02;
	Cyclic#2.::gHardWare.DOF322_1[2] AT %QX."X20DOF322_A".DigitalOutput03;
	Cyclic#2.::gHardWare.DOF322_1[3] AT %QX."X20DOF322_A".DigitalOutput04;
	Cyclic#2.::gHardWare.DOF322_1[4] AT %QX."X20DOF322_A".DigitalOutput05;
	Cyclic#2.::gHardWare.DOF322_1[5] AT %QX."X20DOF322_A".DigitalOutput06;
	Cyclic#2.::gHardWare.DOF322_1[6] AT %QX."X20DOF322_A".DigitalOutput07;
	Cyclic#2.::gHardWare.DOF322_1[7] AT %QX."X20DOF322_A".DigitalOutput08;
	Cyclic#2.::gHardWare.DOF322_1[8] AT %QX."X20DOF322_A".DigitalOutput09;
	Cyclic#2.::gHardWare.DOF322_1[9] AT %QX."X20DOF322_A".DigitalOutput10;
	Cyclic#2.::gHardWare.DOF322_1[10] AT %QX."X20DOF322_A".DigitalOutput11;
	Cyclic#2.::gHardWare.DOF322_1[11] AT %QX."X20DOF322_A".DigitalOutput12;
	Cyclic#2.::gHardWare.DOF322_1[12] AT %QX."X20DOF322_A".DigitalOutput13;
	Cyclic#2.::gHardWare.DOF322_1[13] AT %QX."X20DOF322_A".DigitalOutput14;
	Cyclic#2.::gHardWare.DOF322_1[14] AT %QX."X20DOF322_A".DigitalOutput15;
	Cyclic#2.::gHardWare.DOF322_1[15] AT %QX."X20DOF322_A".DigitalOutput16;
	Cyclic#2.::gHardWare.ModuleOk.DOF322_2 AT %IX."X20DOF322_B".ModuleOk;
	Cyclic#2.::gHardWare.DOF322_2[0] AT %QX."X20DOF322_B".DigitalOutput01;
	Cyclic#2.::gHardWare.DOF322_2[1] AT %QX."X20DOF322_B".DigitalOutput02;
	Cyclic#2.::gHardWare.DOF322_2[2] AT %QX."X20DOF322_B".DigitalOutput03;
	Cyclic#2.::gHardWare.DOF322_2[3] AT %QX."X20DOF322_B".DigitalOutput04;
	Cyclic#2.::gHardWare.DOF322_2[4] AT %QX."X20DOF322_B".DigitalOutput05;
	Cyclic#2.::gHardWare.DOF322_2[5] AT %QX."X20DOF322_B".DigitalOutput06;
	Cyclic#2.::gHardWare.DOF322_2[6] AT %QX."X20DOF322_B".DigitalOutput07;
	Cyclic#2.::gHardWare.DOF322_2[7] AT %QX."X20DOF322_B".DigitalOutput08;
	Cyclic#2.::gHardWare.DOF322_2[8] AT %QX."X20DOF322_B".DigitalOutput09;
	Cyclic#2.::gHardWare.DOF322_2[9] AT %QX."X20DOF322_B".DigitalOutput10;
	Cyclic#2.::gHardWare.DOF322_2[10] AT %QX."X20DOF322_B".DigitalOutput11;
	Cyclic#2.::gHardWare.DOF322_2[11] AT %QX."X20DOF322_B".DigitalOutput12;
	Cyclic#2.::gHardWare.DOF322_2[12] AT %QX."X20DOF322_B".DigitalOutput13;
	Cyclic#2.::gHardWare.DOF322_2[13] AT %QX."X20DOF322_B".DigitalOutput14;
	Cyclic#2.::gHardWare.DOF322_2[14] AT %QX."X20DOF322_B".DigitalOutput15;
	Cyclic#2.::gHardWare.DOF322_2[15] AT %QX."X20DOF322_B".DigitalOutput16;
	Cyclic#2.::gHardWare.ModuleOk.DOF322_3 AT %IX."X20DOF322_C".ModuleOk;
	Cyclic#2.::gHardWare.DOF322_3[0] AT %QX."X20DOF322_C".DigitalOutput01;
	Cyclic#2.::gHardWare.DOF322_3[1] AT %QX."X20DOF322_C".DigitalOutput02;
	Cyclic#2.::gHardWare.DOF322_3[2] AT %QX."X20DOF322_C".DigitalOutput03;
	Cyclic#2.::gHardWare.DOF322_3[3] AT %QX."X20DOF322_C".DigitalOutput04;
	Cyclic#2.::gHardWare.DOF322_3[4] AT %QX."X20DOF322_C".DigitalOutput05;
	Cyclic#2.::gHardWare.DOF322_3[5] AT %QX."X20DOF322_C".DigitalOutput06;
	Cyclic#2.::gHardWare.DOF322_3[6] AT %QX."X20DOF322_C".DigitalOutput07;
	Cyclic#2.::gHardWare.DOF322_3[7] AT %QX."X20DOF322_C".DigitalOutput08;
	Cyclic#2.::gHardWare.DOF322_3[8] AT %QX."X20DOF322_C".DigitalOutput09;
	Cyclic#2.::gHardWare.DOF322_3[9] AT %QX."X20DOF322_C".DigitalOutput10;
	Cyclic#2.::gHardWare.DOF322_3[10] AT %QX."X20DOF322_C".DigitalOutput11;
	Cyclic#2.::gHardWare.DOF322_3[11] AT %QX."X20DOF322_C".DigitalOutput12;
	Cyclic#2.::gHardWare.DOF322_3[12] AT %QX."X20DOF322_C".DigitalOutput13;
	Cyclic#2.::gHardWare.DOF322_3[13] AT %QX."X20DOF322_C".DigitalOutput14;
	Cyclic#2.::gHardWare.DOF322_3[14] AT %QX."X20DOF322_C".DigitalOutput15;
	Cyclic#2.::gHardWare.DOF322_3[15] AT %QX."X20DOF322_C".DigitalOutput16;
	Cyclic#2.::gHardWare.ModuleOk.DOF322_4 AT %IX."X20DOF322_D".ModuleOk;
	Cyclic#2.::gHardWare.DOF322_4[0] AT %QX."X20DOF322_D".DigitalOutput01;
	Cyclic#2.::gHardWare.DOF322_4[1] AT %QX."X20DOF322_D".DigitalOutput02;
	Cyclic#2.::gHardWare.DOF322_4[2] AT %QX."X20DOF322_D".DigitalOutput03;
	Cyclic#2.::gHardWare.DOF322_4[3] AT %QX."X20DOF322_D".DigitalOutput04;
	Cyclic#2.::gHardWare.DOF322_4[4] AT %QX."X20DOF322_D".DigitalOutput05;
	Cyclic#2.::gHardWare.DOF322_4[5] AT %QX."X20DOF322_D".DigitalOutput06;
	Cyclic#2.::gHardWare.DOF322_4[6] AT %QX."X20DOF322_D".DigitalOutput07;
	Cyclic#2.::gHardWare.DOF322_4[7] AT %QX."X20DOF322_D".DigitalOutput08;
	Cyclic#2.::gHardWare.DOF322_4[8] AT %QX."X20DOF322_D".DigitalOutput09;
	Cyclic#2.::gHardWare.DOF322_4[9] AT %QX."X20DOF322_D".DigitalOutput10;
	Cyclic#2.::gHardWare.DOF322_4[10] AT %QX."X20DOF322_D".DigitalOutput11;
	Cyclic#2.::gHardWare.DOF322_4[11] AT %QX."X20DOF322_D".DigitalOutput12;
	Cyclic#2.::gHardWare.DOF322_4[12] AT %QX."X20DOF322_D".DigitalOutput13;
	Cyclic#2.::gHardWare.DOF322_4[13] AT %QX."X20DOF322_D".DigitalOutput14;
	Cyclic#2.::gHardWare.DOF322_4[14] AT %QX."X20DOF322_D".DigitalOutput15;
	Cyclic#2.::gHardWare.DOF322_4[15] AT %QX."X20DOF322_D".DigitalOutput16;
	Cyclic#2.::gHardWare.ModuleOk.DOF322_5 AT %IX."X20DOF322_E".ModuleOk;
	Cyclic#2.::gHardWare.DOF322_5[0] AT %QX."X20DOF322_E".DigitalOutput01;
	Cyclic#2.::gHardWare.DOF322_5[1] AT %QX."X20DOF322_E".DigitalOutput02;
	Cyclic#2.::gHardWare.DOF322_5[2] AT %QX."X20DOF322_E".DigitalOutput03;
	Cyclic#2.::gHardWare.DOF322_5[3] AT %QX."X20DOF322_E".DigitalOutput04;
	Cyclic#2.::gHardWare.DOF322_5[4] AT %QX."X20DOF322_E".DigitalOutput05;
	Cyclic#2.::gHardWare.DOF322_5[5] AT %QX."X20DOF322_E".DigitalOutput06;
	Cyclic#2.::gHardWare.DOF322_5[6] AT %QX."X20DOF322_E".DigitalOutput07;
	Cyclic#2.::gHardWare.DOF322_5[7] AT %QX."X20DOF322_E".DigitalOutput08;
	Cyclic#2.::gHardWare.DOF322_5[8] AT %QX."X20DOF322_E".DigitalOutput09;
	Cyclic#2.::gHardWare.DOF322_5[9] AT %QX."X20DOF322_E".DigitalOutput10;
	Cyclic#2.::gHardWare.DOF322_5[10] AT %QX."X20DOF322_E".DigitalOutput11;
	Cyclic#2.::gHardWare.DOF322_5[11] AT %QX."X20DOF322_E".DigitalOutput12;
	Cyclic#2.::gHardWare.DOF322_5[12] AT %QX."X20DOF322_E".DigitalOutput13;
	Cyclic#2.::gHardWare.DOF322_5[13] AT %QX."X20DOF322_E".DigitalOutput14;
	Cyclic#2.::gHardWare.DOF322_5[14] AT %QX."X20DOF322_E".DigitalOutput15;
	Cyclic#2.::gHardWare.DOF322_5[15] AT %QX."X20DOF322_E".DigitalOutput16;
	Cyclic#2.::gHardWare.ModuleOk.DO8332_1 AT %IX."X20DO8332_A".ModuleOk;
	Cyclic#2.::gHardWare.DO8332_1[0] AT %QX."X20DO8332_A".DigitalOutput01;
	Cyclic#2.::gHardWare.DO8332_1[1] AT %QX."X20DO8332_A".DigitalOutput02;
	Cyclic#2.::gHardWare.DO8332_1[2] AT %QX."X20DO8332_A".DigitalOutput03;
	Cyclic#2.::gHardWare.DO8332_1[3] AT %QX."X20DO8332_A".DigitalOutput04;
	Cyclic#2.::gHardWare.DO8332_1[4] AT %QX."X20DO8332_A".DigitalOutput05;
	Cyclic#2.::gHardWare.DO8332_1[5] AT %QX."X20DO8332_A".DigitalOutput06;
	Cyclic#2.::gHardWare.DO8332_1[6] AT %QX."X20DO8332_A".DigitalOutput07;
	Cyclic#2.::gHardWare.DO8332_1[7] AT %QX."X20DO8332_A".DigitalOutput08;
	Cyclic#2.::gHardWare.ModuleOk.DO8332_2 AT %IX."X20DO8332_B".ModuleOk;
	Cyclic#2.::gHardWare.DO8332_2[0] AT %QX."X20DO8332_B".DigitalOutput01;
	Cyclic#2.::gHardWare.DO8332_2[1] AT %QX."X20DO8332_B".DigitalOutput02;
	Cyclic#2.::gHardWare.DO8332_2[2] AT %QX."X20DO8332_B".DigitalOutput03;
	Cyclic#2.::gHardWare.DO8332_2[3] AT %QX."X20DO8332_B".DigitalOutput04;
	Cyclic#2.::gHardWare.DO8332_2[4] AT %QX."X20DO8332_B".DigitalOutput05;
	Cyclic#2.::gHardWare.DO8332_2[5] AT %QX."X20DO8332_B".DigitalOutput06;
	Cyclic#2.::gHardWare.DO8332_2[6] AT %QX."X20DO8332_B".DigitalOutput07;
	Cyclic#2.::gHardWare.DO8332_2[7] AT %QX."X20DO8332_B".DigitalOutput08;
	Cyclic#2.::gHardWare.ModuleOk.DO8332_3 AT %IX."X20DO8332_C".ModuleOk;
	Cyclic#2.::gHardWare.DO8332_3[0] AT %QX."X20DO8332_C".DigitalOutput01;
	Cyclic#2.::gHardWare.DO8332_3[1] AT %QX."X20DO8332_C".DigitalOutput02;
	Cyclic#2.::gHardWare.DO8332_3[2] AT %QX."X20DO8332_C".DigitalOutput03;
	Cyclic#2.::gHardWare.DO8332_3[3] AT %QX."X20DO8332_C".DigitalOutput04;
	Cyclic#2.::gHardWare.DO8332_3[4] AT %QX."X20DO8332_C".DigitalOutput05;
	Cyclic#2.::gHardWare.DO8332_3[5] AT %QX."X20DO8332_C".DigitalOutput06;
	Cyclic#2.::gHardWare.DO8332_3[6] AT %QX."X20DO8332_C".DigitalOutput07;
	Cyclic#2.::gHardWare.DO8332_3[7] AT %QX."X20DO8332_C".DigitalOutput08;
	Cyclic#2.::gHardWare.ModuleOk.DO8332_4 AT %IX."X20DO8332_D".ModuleOk;
	Cyclic#2.::gHardWare.DO8332_4[0] AT %QX."X20DO8332_D".DigitalOutput01;
	Cyclic#2.::gHardWare.DO8332_4[1] AT %QX."X20DO8332_D".DigitalOutput02;
	Cyclic#2.::gHardWare.DO8332_4[2] AT %QX."X20DO8332_D".DigitalOutput03;
	Cyclic#2.::gHardWare.DO8332_4[3] AT %QX."X20DO8332_D".DigitalOutput04;
	Cyclic#2.::gHardWare.DO8332_4[4] AT %QX."X20DO8332_D".DigitalOutput05;
	Cyclic#2.::gHardWare.DO8332_4[5] AT %QX."X20DO8332_D".DigitalOutput06;
	Cyclic#2.::gHardWare.DO8332_4[6] AT %QX."X20DO8332_D".DigitalOutput07;
	Cyclic#2.::gHardWare.DO8332_4[7] AT %QX."X20DO8332_D".DigitalOutput08;
	Cyclic#2.::gHardWare.ModuleOk.PS3300_1 AT %IX."X20PS3300".ModuleOk;
	Cyclic#2.::gHardWare.ModuleOk.AI4632_1 AT %IX."X20AI4632_A".ModuleOk;
	Cyclic#1.::gHardWare.AI4632_1[0] AT %IW."X20AI4632_A".AnalogInput01;
	Cyclic#1.::gHardWare.AI4632_1[1] AT %IW."X20AI4632_A".AnalogInput02;
	Cyclic#1.::gHardWare.AI4632_1[2] AT %IW."X20AI4632_A".AnalogInput03;
	Cyclic#1.::gHardWare.AI4632_1[3] AT %IW."X20AI4632_A".AnalogInput04;
	Cyclic#2.::gHardWare.ModuleOk.AI4632_2 AT %IX."X20AI4632_B".ModuleOk;
	Cyclic#1.::gHardWare.AI4632_2[0] AT %IW."X20AI4632_B".AnalogInput01;
	Cyclic#1.::gHardWare.AI4632_2[1] AT %IW."X20AI4632_B".AnalogInput02;
	Cyclic#1.::gHardWare.AI4632_2[2] AT %IW."X20AI4632_B".AnalogInput03;
	Cyclic#1.::gHardWare.AI4632_2[3] AT %IW."X20AI4632_B".AnalogInput04;
	Cyclic#2.::gHardWare.ModuleOk.AO4622_1 AT %IX."X20AO4622_A".ModuleOk;
	Cyclic#1.::gHardWare.AO4622_1[0] AT %QW."X20AO4622_A".AnalogOutput01;
	Cyclic#1.::gHardWare.AO4622_1[1] AT %QW."X20AO4622_A".AnalogOutput02;
	Cyclic#1.::gHardWare.AO4622_1[2] AT %QW."X20AO4622_A".AnalogOutput03;
	Cyclic#1.::gHardWare.AO4622_1[3] AT %QW."X20AO4622_A".AnalogOutput04;
	Cyclic#2.::gHardWare.ModuleOk.AO4622_2 AT %IX."X20AO4622_B".ModuleOk;
	Cyclic#1.::gHardWare.AO4622_2[0] AT %QW."X20AO4622_B".AnalogOutput01;
	Cyclic#1.::gHardWare.AO4622_2[1] AT %QW."X20AO4622_B".AnalogOutput02;
	Cyclic#1.::gHardWare.AO4622_2[2] AT %QW."X20AO4622_B".AnalogOutput03;
	Cyclic#1.::gHardWare.AO4622_2[3] AT %QW."X20AO4622_B".AnalogOutput04;
	Cyclic#2.gHardWare.ModuleOk.AP3131_1 AT %IX."X20AP3131_A".ModuleOk;
	Cyclic#3.gHardWare.AP3131_1.IrmsA AT %IW."X20AP3131_A".IrmsA;
	Cyclic#3.gHardWare.AP3131_1.IrmsB AT %IW."X20AP3131_A".IrmsB;
	Cyclic#3.gHardWare.AP3131_1.IrmsC AT %IW."X20AP3131_A".IrmsC;
	Cyclic#3.::gHardWare.AP3131_1.PmeanT AT %IW."X20AP3131_A".PmeanT;
	Cyclic#3.::gHardWare.AP3131_1.SmeanT AT %IW."X20AP3131_A".SmeanT;
	Cyclic#3.::gHardWare.AP3131_1.PFmeanT AT %IW."X20AP3131_A".PFmeanT;
	Cyclic#3.::gHardWare.AP3131_1.AenergyT AT %ID."X20AP3131_A".AenergyT;
	Cyclic#3.::gHardWare.AP3131_1.SAenergyT AT %ID."X20AP3131_A".SAenergyT;
	Cyclic#2.::gHardWare.AP3131_1.TrigDFT AT %QX."X20AP3131_A".TrigDFT;
	Cyclic#2.::gHardWare.AP3131_1.EnableEnergy AT %QX."X20AP3131_A".EnabEnergy;
	Cyclic#2.::gHardWare.AP3131_1.ClearEnergy AT %QX."X20AP3131_A".ClearEnergy;
	Cyclic#2.::gHardWare.AP3131_1.TrigForceEnergy AT %QX."X20AP3131_A".ForceEnergy;
	Cyclic#2.gHardWare.ModuleOk.AP3131_2 AT %IX."X20AP3131_B".ModuleOk;
	Cyclic#3.::gHardWare.AP3131_2.IrmsA AT %IW."X20AP3131_B".IrmsA;
	Cyclic#3.::gHardWare.AP3131_2.IrmsB AT %IW."X20AP3131_B".IrmsB;
	Cyclic#3.::gHardWare.AP3131_2.IrmsC AT %IW."X20AP3131_B".IrmsC;
	Cyclic#3.::gHardWare.AP3131_2.PmeanT AT %IW."X20AP3131_B".PmeanT;
	Cyclic#3.::gHardWare.AP3131_2.SmeanT AT %IW."X20AP3131_B".SmeanT;
	Cyclic#3.::gHardWare.AP3131_2.PFmeanT AT %IW."X20AP3131_B".PFmeanT;
	Cyclic#3.::gHardWare.AP3131_2.AenergyT AT %ID."X20AP3131_B".AenergyT;
	Cyclic#3.::gHardWare.AP3131_2.SAenergyT AT %ID."X20AP3131_B".SAenergyT;
	Cyclic#2.::gHardWare.AP3131_2.TrigDFT AT %QX."X20AP3131_B".TrigDFT;
	Cyclic#2.::gHardWare.AP3131_2.EnableEnergy AT %QX."X20AP3131_B".EnabEnergy;
	Cyclic#2.::gHardWare.AP3131_2.ClearEnergy AT %QX."X20AP3131_B".ClearEnergy;
	Cyclic#2.::gHardWare.AP3131_2.TrigForceEnergy AT %QX."X20AP3131_B".ForceEnergy;
	Cyclic#2.gHardWare.ModuleOk.AP3131_3 AT %IX."X20AP3131_C".ModuleOk;
	Cyclic#3.::gHardWare.AP3131_3.IrmsA AT %IW."X20AP3131_C".IrmsA;
	Cyclic#3.::gHardWare.AP3131_3.IrmsB AT %IW."X20AP3131_C".IrmsB;
	Cyclic#3.::gHardWare.AP3131_3.IrmsC AT %IW."X20AP3131_C".IrmsC;
	Cyclic#3.::gHardWare.AP3131_3.PmeanT AT %IW."X20AP3131_C".PmeanT;
	Cyclic#3.::gHardWare.AP3131_3.SmeanT AT %IW."X20AP3131_C".SmeanT;
	Cyclic#3.::gHardWare.AP3131_3.PFmeanT AT %IW."X20AP3131_C".PFmeanT;
	Cyclic#3.::gHardWare.AP3131_3.AenergyT AT %ID."X20AP3131_C".AenergyT;
	Cyclic#3.::gHardWare.AP3131_3.SAenergyT AT %ID."X20AP3131_C".SAenergyT;
	Cyclic#2.::gHardWare.AP3131_3.TrigDFT AT %QX."X20AP3131_C".TrigDFT;
	Cyclic#2.::gHardWare.AP3131_3.EnableEnergy AT %QX."X20AP3131_C".EnabEnergy;
	Cyclic#2.::gHardWare.AP3131_3.ClearEnergy AT %QX."X20AP3131_C".ClearEnergy;
	Cyclic#2.::gHardWare.AP3131_3.TrigForceEnergy AT %QX."X20AP3131_C".ForceEnergy;
	Cyclic#2.gHardWare.ModuleOk.ATC402_1 AT %IX."X20ATC402_A".ModuleOk;
	Cyclic#2.gHardWare.ATC402_1[0] AT %IW."X20ATC402_A".Temperature01;
	Cyclic#2.gHardWare.ATC402_1[1] AT %IW."X20ATC402_A".Temperature02;
	Cyclic#2.gHardWare.ATC402_1[2] AT %IW."X20ATC402_A".Temperature03;
	Cyclic#2.gHardWare.ATC402_1[3] AT %IW."X20ATC402_A".Temperature04;
	Cyclic#2.gHardWare.ATC402_1[4] AT %IW."X20ATC402_A".Temperature05;
	Cyclic#2.gHardWare.ATC402_1[5] AT %IW."X20ATC402_A".Temperature06;
	Cyclic#2.::gHardWare.ModuleOk.ATC402_2 AT %IX."X20ATC402_B".ModuleOk;
	Cyclic#2.::gHardWare.ATC402_2[0] AT %IW."X20ATC402_B".Temperature01;
	Cyclic#2.gHardWare.ATC402_2[1] AT %IW."X20ATC402_B".Temperature02;
	Cyclic#2.gHardWare.ATC402_2[2] AT %IW."X20ATC402_B".Temperature03;
	Cyclic#2.gHardWare.ATC402_2[3] AT %IW."X20ATC402_B".Temperature04;
	Cyclic#2.gHardWare.ATC402_2[4] AT %IW."X20ATC402_B".Temperature05;
	Cyclic#2.gHardWare.ATC402_2[5] AT %IW."X20ATC402_B".Temperature06;
	Cyclic#2.gHardWare.ModuleOk.ATC402_3 AT %IX."X20ATC402_C".ModuleOk;
	Cyclic#2.gHardWare.ATC402_3[0] AT %IW."X20ATC402_C".Temperature01;
	Cyclic#2.gHardWare.ATC402_3[1] AT %IW."X20ATC402_C".Temperature02;
	Cyclic#2.gHardWare.ATC402_3[2] AT %IW."X20ATC402_C".Temperature03;
	Cyclic#2.gHardWare.ATC402_3[3] AT %IW."X20ATC402_C".Temperature04;
	Cyclic#2.gHardWare.ATC402_3[4] AT %IW."X20ATC402_C".Temperature05;
	Cyclic#2.gHardWare.ATC402_3[5] AT %IW."X20ATC402_C".Temperature06;
	Cyclic#2.gHardWare.ModuleOk.ATC402_4 AT %IX."X20ATC402_D".ModuleOk;
	Cyclic#2.gHardWare.ATC402_4[0] AT %IW."X20ATC402_D".Temperature01;
	Cyclic#2.gHardWare.ATC402_4[1] AT %IW."X20ATC402_D".Temperature02;
	Cyclic#2.gHardWare.ATC402_4[2] AT %IW."X20ATC402_D".Temperature03;
	Cyclic#2.gHardWare.ATC402_4[3] AT %IW."X20ATC402_D".Temperature04;
	Cyclic#2.gHardWare.ATC402_4[4] AT %IW."X20ATC402_D".Temperature05;
	Cyclic#2.gHardWare.ATC402_4[5] AT %IW."X20ATC402_D".Temperature06;
	Cyclic#2.gHardWare.ModuleOk.ATC402_5 AT %IX."X20ATC402_E".ModuleOk;
	Cyclic#2.gHardWare.ATC402_5[0] AT %IW."X20ATC402_E".Temperature01;
	Cyclic#2.gHardWare.ATC402_5[1] AT %IW."X20ATC402_E".Temperature02;
	Cyclic#2.gHardWare.ATC402_5[2] AT %IW."X20ATC402_E".Temperature03;
	Cyclic#2.gHardWare.ATC402_5[3] AT %IW."X20ATC402_E".Temperature04;
	Cyclic#2.gHardWare.ATC402_5[4] AT %IW."X20ATC402_E".Temperature05;
	Cyclic#2.gHardWare.ATC402_5[5] AT %IW."X20ATC402_E".Temperature06;
	::gHardWare.ModuleOk.PS9400_2 AT %IX."X20PS9400a".ModuleOk;
	::gHardWare.ModuleOk.BC0083_2 AT %IX."X20BC0083a".ModuleOk;
	Cyclic#2.::gExtruderACtrl.InverterStatus.bSwitchOn AT %IX."8I84xxxxxxx.01P-1".ETAD_Input_Bool_01;
	Cyclic#2.::gExtruderACtrl.InverterStatus.ActSpeed AT %IW."8I84xxxxxxx.01P-1".RFRD_Input;
	Cyclic#2.::gExtruderACtrl.InverterStatus.ActTorque AT %IW."8I84xxxxxxx.01P-1".OTR_Input;
	Cyclic#2.::gExtruderACtrl.InverterStatus.Current AT %IW."8I84xxxxxxx.01P-1".LCR_Input;
	Cyclic#2.::gExtruderACtrl.InverterCmd.bSwitchOn AT %QX."8I84xxxxxxx.01P-1".CMDD_Output_Bool_00;
	Cyclic#2.::gExtruderACtrl.InverterCmd.bEnableCtrl AT %QX."8I84xxxxxxx.01P-1".CMDD_Output_Bool_03;
	Cyclic#2.::gExtruderACtrl.InverterCmd.bAskStop AT %QX."8I84xxxxxxx.01P-1".CMDD_Output_Bool_08;
	Cyclic#2.::gExtruderACtrl.InverterCmd.bInverse AT %QX."8I84xxxxxxx.01P-1".CMDD_Output_Bool_11;
	Cyclic#2.::gExtruderACtrl.SetSpeed AT %QW."8I84xxxxxxx.01P-1".LFRD_Output;
	Cyclic#2.::gExtruderACtrl.InverterStatus.bModuleOk AT %IX."8I84xxxxxxx.01P-1".ModuleOk;
	Cyclic#2.::gExtruderACtrl.InverterStatus.bRunning AT %IX."8I84xxxxxxx.01P-1".ETAD_Input_Bool_02;
	Cyclic#2.::gExtruderACtrl.InverterStatus.bWarningOrAlarm AT %IX."8I84xxxxxxx.01P-1".ETAD_Input_Bool_07;
	Cyclic#2.::gExtruderACtrl.InverterStatus.DriverTemp AT %IW."8I84xxxxxxx.01P-1".THD_Input;
	Cyclic#2.::gExtruderACtrl.InverterStatus.MotorTemp AT %IW."8I84xxxxxxx.01P-1".THR_Input;
	Cyclic#2.::gExtruderACtrl.InverterStatus.FaultID AT %IW."8I84xxxxxxx.01P-1".LFT_Input;
	Cyclic#2.::gExtruderACtrl.InverterStatus.bModuleOk AT %QX."8I84xxxxxxx.01P-1".CMDD_Output_Bool_02;
	Cyclic#2.::gExtruderACtrl.InverterStatus.bModuleOk AT %QX."8I84xxxxxxx.01P-1".CMDD_Output_Bool_01;
	Cyclic#2.::gExtruderACtrl.InverterCmd.bResetFault AT %QX."8I84xxxxxxx.01P-1".CMDD_Output_Bool_07;
	Cyclic#2.::gExtruderACtrl.InverterCmd.bSpeed32767 AT %QX."8I84xxxxxxx.01P-1".CMI_Output_Bool_09;
	Cyclic#2.::gExtruderACtrl.SetTorque AT %QW."8I84xxxxxxx.01P-1".LTR_Output;
	Cyclic#2.::gExtruderACtrl.InverterStatus.PowerOnReady AT %IX."8I84xxxxxxx.01P-1".ETAD_Input_Bool_00;
	Cyclic#2.::gExtruderBCtrl.InverterStatus.bModuleOk AT %IX."8I84xxxxxxx.01P-1a".ModuleOk;
	Cyclic#2.::gExtruderBCtrl.InverterStatus.PowerOnReady AT %IX."8I84xxxxxxx.01P-1a".ETAD_Input_Bool_00;
	Cyclic#2.::gExtruderBCtrl.InverterStatus.bSwitchOn AT %IX."8I84xxxxxxx.01P-1a".ETAD_Input_Bool_01;
	Cyclic#2.::gExtruderBCtrl.InverterStatus.bRunning AT %IX."8I84xxxxxxx.01P-1a".ETAD_Input_Bool_02;
	Cyclic#2.::gExtruderBCtrl.InverterStatus.bWarningOrAlarm AT %IX."8I84xxxxxxx.01P-1a".ETAD_Input_Bool_07;
	Cyclic#2.::gExtruderBCtrl.InverterStatus.ActSpeed AT %IW."8I84xxxxxxx.01P-1a".RFRD_Input;
	Cyclic#2.::gExtruderBCtrl.InverterStatus.ActTorque AT %IW."8I84xxxxxxx.01P-1a".OTR_Input;
	Cyclic#2.::gExtruderBCtrl.InverterStatus.Current AT %IW."8I84xxxxxxx.01P-1a".LCR_Input;
	Cyclic#2.::gExtruderBCtrl.InverterStatus.DriverTemp AT %IW."8I84xxxxxxx.01P-1a".THD_Input;
	Cyclic#2.::gExtruderBCtrl.InverterStatus.MotorTemp AT %IW."8I84xxxxxxx.01P-1a".THR_Input;
	Cyclic#2.::gExtruderBCtrl.InverterStatus.FaultID AT %IW."8I84xxxxxxx.01P-1a".LFT_Input;
	Cyclic#2.::gExtruderBCtrl.InverterCmd.bSwitchOn AT %QX."8I84xxxxxxx.01P-1a".CMDD_Output_Bool_00;
	Cyclic#2.::gExtruderBCtrl.InverterStatus.bModuleOk AT %QX."8I84xxxxxxx.01P-1a".CMDD_Output_Bool_01;
	Cyclic#2.::gExtruderBCtrl.InverterStatus.bModuleOk AT %QX."8I84xxxxxxx.01P-1a".CMDD_Output_Bool_02;
	Cyclic#2.::gExtruderBCtrl.InverterCmd.bEnableCtrl AT %QX."8I84xxxxxxx.01P-1a".CMDD_Output_Bool_03;
	Cyclic#2.::gExtruderBCtrl.InverterCmd.bResetFault AT %QX."8I84xxxxxxx.01P-1a".CMDD_Output_Bool_07;
	Cyclic#2.::gExtruderBCtrl.InverterCmd.bAskStop AT %QX."8I84xxxxxxx.01P-1a".CMDD_Output_Bool_08;
	Cyclic#2.::gExtruderBCtrl.InverterCmd.bInverse AT %QX."8I84xxxxxxx.01P-1a".CMDD_Output_Bool_11;
	Cyclic#2.::gExtruderBCtrl.InverterCmd.bSpeed32767 AT %QX."8I84xxxxxxx.01P-1a".CMI_Output_Bool_09;
	Cyclic#2.::gExtruderBCtrl.SetSpeed AT %QW."8I84xxxxxxx.01P-1a".LFRD_Output;
	Cyclic#2.::gExtruderBCtrl.SetTorque AT %QW."8I84xxxxxxx.01P-1a".LTR_Output;
	Cyclic#2.::gExtruderCCtrl.InverterStatus.bModuleOk AT %IX."8I84xxxxxxx.01P-1b".ModuleOk;
	Cyclic#2.::gExtruderCCtrl.InverterStatus.PowerOnReady AT %IX."8I84xxxxxxx.01P-1b".ETAD_Input_Bool_00;
	Cyclic#2.::gExtruderCCtrl.InverterStatus.bSwitchOn AT %IX."8I84xxxxxxx.01P-1b".ETAD_Input_Bool_01;
	Cyclic#2.::gExtruderCCtrl.InverterStatus.bRunning AT %IX."8I84xxxxxxx.01P-1b".ETAD_Input_Bool_02;
	Cyclic#2.::gExtruderCCtrl.InverterStatus.bWarningOrAlarm AT %IX."8I84xxxxxxx.01P-1b".ETAD_Input_Bool_07;
	Cyclic#2.::gExtruderCCtrl.InverterStatus.ActSpeed AT %IW."8I84xxxxxxx.01P-1b".RFRD_Input;
	Cyclic#2.::gExtruderCCtrl.InverterStatus.ActTorque AT %IW."8I84xxxxxxx.01P-1b".OTR_Input;
	Cyclic#2.::gExtruderCCtrl.InverterStatus.Current AT %IW."8I84xxxxxxx.01P-1b".LCR_Input;
	Cyclic#2.::gExtruderCCtrl.InverterStatus.DriverTemp AT %IW."8I84xxxxxxx.01P-1b".THD_Input;
	Cyclic#2.::gExtruderCCtrl.InverterStatus.MotorTemp AT %IW."8I84xxxxxxx.01P-1b".THR_Input;
	Cyclic#2.::gExtruderCCtrl.InverterStatus.FaultID AT %IW."8I84xxxxxxx.01P-1b".LFT_Input;
	Cyclic#2.::gExtruderCCtrl.InverterCmd.bSwitchOn AT %QX."8I84xxxxxxx.01P-1b".CMDD_Output_Bool_00;
	Cyclic#2.::gExtruderCCtrl.InverterStatus.bModuleOk AT %QX."8I84xxxxxxx.01P-1b".CMDD_Output_Bool_01;
	Cyclic#2.::gExtruderCCtrl.InverterStatus.bModuleOk AT %QX."8I84xxxxxxx.01P-1b".CMDD_Output_Bool_02;
	Cyclic#2.::gExtruderCCtrl.InverterCmd.bEnableCtrl AT %QX."8I84xxxxxxx.01P-1b".CMDD_Output_Bool_03;
	Cyclic#2.::gExtruderCCtrl.InverterCmd.bResetFault AT %QX."8I84xxxxxxx.01P-1b".CMDD_Output_Bool_07;
	Cyclic#2.::gExtruderCCtrl.InverterCmd.bAskStop AT %QX."8I84xxxxxxx.01P-1b".CMDD_Output_Bool_08;
	Cyclic#2.::gExtruderCCtrl.InverterCmd.bInverse AT %QX."8I84xxxxxxx.01P-1b".CMDD_Output_Bool_11;
	Cyclic#2.::gExtruderCCtrl.InverterCmd.bSpeed32767 AT %QX."8I84xxxxxxx.01P-1b".CMI_Output_Bool_09;
	Cyclic#2.::gExtruderCCtrl.SetSpeed AT %QW."8I84xxxxxxx.01P-1b".LFRD_Output;
	Cyclic#2.::gExtruderCCtrl.SetTorque AT %QW."8I84xxxxxxx.01P-1b".LTR_Output;
	Cyclic#2.::gHardWare.DO8332_5[0] AT %QX."X20DO8332_E".DigitalOutput01;
	Cyclic#2.::gHardWare.ModuleOk.DO8332_5 AT %IX."X20DO8332_E".ModuleOk;
	Cyclic#2.::gHardWare.DO8332_5[1] AT %QX."X20DO8332_E".DigitalOutput02;
	Cyclic#2.::gHardWare.DO8332_5[2] AT %QX."X20DO8332_E".DigitalOutput03;
	Cyclic#2.::gHardWare.DO8332_5[3] AT %QX."X20DO8332_E".DigitalOutput04;
	Cyclic#2.::gHardWare.DO8332_5[4] AT %QX."X20DO8332_E".DigitalOutput05;
	Cyclic#2.::gHardWare.DO8332_5[5] AT %QX."X20DO8332_E".DigitalOutput06;
	Cyclic#2.::gHardWare.DO8332_5[6] AT %QX."X20DO8332_E".DigitalOutput07;
	Cyclic#2.::gHardWare.DO8332_5[7] AT %QX."X20DO8332_E".DigitalOutput08;
	Cyclic#2.::gHardWare.DO8332_6[0] AT %QX."X20DO8332_F".DigitalOutput01;
	Cyclic#2.::gHardWare.DO8332_6[1] AT %QX."X20DO8332_F".DigitalOutput02;
	Cyclic#2.::gHardWare.DO8332_6[2] AT %QX."X20DO8332_F".DigitalOutput03;
	Cyclic#2.::gHardWare.DO8332_6[3] AT %QX."X20DO8332_F".DigitalOutput04;
	Cyclic#2.::gHardWare.DO8332_6[4] AT %QX."X20DO8332_F".DigitalOutput05;
	Cyclic#2.::gHardWare.DO8332_6[5] AT %QX."X20DO8332_F".DigitalOutput06;
	Cyclic#2.::gHardWare.DO8332_6[6] AT %QX."X20DO8332_F".DigitalOutput07;
	Cyclic#2.::gHardWare.DO8332_6[7] AT %QX."X20DO8332_F".DigitalOutput08;
	Cyclic#2.::gHardWare.ModuleOk.DO8332_6 AT %IX."X20DO8332_F".ModuleOk;
	Cyclic#2.::gHardWare.ModuleOk.DO9322_7 AT %IX."X20DO8332_G".ModuleOk;
	Cyclic#2.::gHardWare.ModuleOk.DO8332_8 AT %IX."X20DO8332_H".ModuleOk;
	Cyclic#2.::gHardWare.DO8332_7[0] AT %QX."X20DO8332_G".DigitalOutput01;
	Cyclic#2.::gHardWare.DO8332_7[1] AT %QX."X20DO8332_G".DigitalOutput02;
	Cyclic#2.::gHardWare.DO8332_7[2] AT %QX."X20DO8332_G".DigitalOutput03;
	Cyclic#2.::gHardWare.DO8332_7[3] AT %QX."X20DO8332_G".DigitalOutput04;
	Cyclic#2.::gHardWare.DO8332_7[4] AT %QX."X20DO8332_G".DigitalOutput05;
	Cyclic#2.::gHardWare.DO8332_7[5] AT %QX."X20DO8332_G".DigitalOutput06;
	Cyclic#2.::gHardWare.DO8332_7[6] AT %QX."X20DO8332_G".DigitalOutput07;
	Cyclic#2.::gHardWare.DO8332_7[7] AT %QX."X20DO8332_G".DigitalOutput08;
	Cyclic#2.::gHardWare.DO8332_8[0] AT %QX."X20DO8332_H".DigitalOutput01;
	Cyclic#2.::gHardWare.DO8332_8[1] AT %QX."X20DO8332_H".DigitalOutput02;
	Cyclic#2.::gHardWare.DO8332_8[2] AT %QX."X20DO8332_H".DigitalOutput03;
	Cyclic#2.::gHardWare.DO8332_8[3] AT %QX."X20DO8332_H".DigitalOutput04;
	Cyclic#2.::gHardWare.DO8332_8[4] AT %QX."X20DO8332_H".DigitalOutput05;
	Cyclic#2.::gHardWare.DO8332_8[5] AT %QX."X20DO8332_H".DigitalOutput06;
	Cyclic#2.::gHardWare.DO8332_8[6] AT %QX."X20DO8332_H".DigitalOutput07;
	Cyclic#2.::gHardWare.DO8332_8[7] AT %QX."X20DO8332_H".DigitalOutput08;
	Cyclic#2.::gHardWare.ModuleOk.DOF322_6 AT %IX."X20DOF322_F".ModuleOk;
	Cyclic#2.::gHardWare.DOF322_6[0] AT %QX."X20DOF322_F".DigitalOutput01;
	Cyclic#2.::gHardWare.DOF322_6[1] AT %QX."X20DOF322_F".DigitalOutput02;
	Cyclic#2.::gHardWare.DOF322_6[2] AT %QX."X20DOF322_F".DigitalOutput03;
	Cyclic#2.::gHardWare.DOF322_6[3] AT %QX."X20DOF322_F".DigitalOutput04;
	Cyclic#2.::gHardWare.DOF322_6[4] AT %QX."X20DOF322_F".DigitalOutput05;
	Cyclic#2.::gHardWare.DOF322_6[5] AT %QX."X20DOF322_F".DigitalOutput06;
	Cyclic#2.::gHardWare.DOF322_6[6] AT %QX."X20DOF322_F".DigitalOutput07;
	Cyclic#2.::gHardWare.DOF322_6[7] AT %QX."X20DOF322_F".DigitalOutput08;
	Cyclic#2.::gHardWare.DOF322_6[8] AT %QX."X20DOF322_F".DigitalOutput09;
	Cyclic#2.::gHardWare.DOF322_6[9] AT %QX."X20DOF322_F".DigitalOutput10;
	Cyclic#2.::gHardWare.DOF322_6[10] AT %QX."X20DOF322_F".DigitalOutput11;
	Cyclic#2.::gHardWare.DOF322_6[11] AT %QX."X20DOF322_F".DigitalOutput12;
	Cyclic#2.::gHardWare.DOF322_6[13] AT %QX."X20DOF322_F".DigitalOutput14;
	Cyclic#2.::gHardWare.DOF322_6[14] AT %QX."X20DOF322_F".DigitalOutput15;
	Cyclic#2.::gHardWare.DOF322_6[15] AT %QX."X20DOF322_F".DigitalOutput16;
	Cyclic#2.::gHardWare.DOF322_6[12] AT %QX."X20DOF322_F".DigitalOutput13;
	Cyclic#2.::gHardWare.ModuleOk.DIF371_4 AT %IX."X20DIF371_D".ModuleOk;
	Cyclic#2.::gHardWare.ModuleOk.ATC402_6 AT %IX."X20ATC402_F".ModuleOk;
	Cyclic#2.::gHardWare.ATC402_6[0] AT %IW."X20ATC402_F".Temperature01;
	Cyclic#2.::gHardWare.ATC402_6[1] AT %IW."X20ATC402_F".Temperature02;
	Cyclic#2.::gHardWare.ATC402_6[2] AT %IW."X20ATC402_F".Temperature03;
	Cyclic#2.::gHardWare.ATC402_6[3] AT %IW."X20ATC402_F".Temperature04;
	Cyclic#2.::gHardWare.ATC402_6[4] AT %IW."X20ATC402_F".Temperature05;
	Cyclic#2.::gHardWare.ATC402_6[5] AT %IW."X20ATC402_F".Temperature06;
	Cyclic#2.::gHardWare.XP0101_1[0] AT %IX."4XP0101.00-00B".DigitalInput01;
	Cyclic#2.::gHardWare.XP0101_1[1] AT %IX."4XP0101.00-00B".DigitalInput02;
	Cyclic#2.::gHardWare.XP0101_1[2] AT %IX."4XP0101.00-00B".DigitalInput03;
	Cyclic#2.::gHardWare.XP0101_1[3] AT %IX."4XP0101.00-00B".DigitalInput04;
	Cyclic#2.::gHardWare.XP0101_1[4] AT %IX."4XP0101.00-00B".DigitalInput05;
	Cyclic#2.::gHardWare.XP0101_1[5] AT %IX."4XP0101.00-00B".DigitalInput06;
	Cyclic#2.::gHardWare.XP0101_1[6] AT %IX."4XP0101.00-00B".DigitalInput07;
	Cyclic#2.::gHardWare.XP0101_1[7] AT %IX."4XP0101.00-00B".DigitalInput08;
	Cyclic#2.::gHardWare.ModuleOk.XP0101_1 AT %IX."4XP0101.00-00B".ModuleOk;
	Cyclic#2.::gHardWare.XP0101Led_1[0] AT %QX."4XP0101.00-00B".DigitalOutput01;
	Cyclic#2.::gHardWare.XP0101Led_1[1] AT %QX."4XP0101.00-00B".DigitalOutput02;
	Cyclic#2.::gHardWare.XP0101Led_1[2] AT %QX."4XP0101.00-00B".DigitalOutput03;
	Cyclic#2.::gHardWare.XP0101Led_1[3] AT %QX."4XP0101.00-00B".DigitalOutput04;
	Cyclic#2.::gHardWare.XP0101Led_1[4] AT %QX."4XP0101.00-00B".DigitalOutput05;
	Cyclic#2.::gHardWare.XP0101Led_1[5] AT %QX."4XP0101.00-00B".DigitalOutput06;
	Cyclic#2.::gHardWare.XP0101Led_1[6] AT %QX."4XP0101.00-00B".DigitalOutput07;
	Cyclic#2.::gHardWare.XP0101Led_1[7] AT %QX."4XP0101.00-00B".DigitalOutput08;
	Cyclic#2.::gHardWare.XP0101Led_1[8] AT %QX."4XP0101.00-00B".DigitalOutput09;
	Cyclic#2.::gHardWare.XP0101Led_1[9] AT %QX."4XP0101.00-00B".DigitalOutput10;
	Cyclic#2.::gHardWare.XP0101Led_1[10] AT %QX."4XP0101.00-00B".DigitalOutput11;
	Cyclic#2.::gHardWare.XP0101Led_1[11] AT %QX."4XP0101.00-00B".DigitalOutput12;
	Cyclic#2.::gHardWare.XP0101Led_1[12] AT %QX."4XP0101.00-00B".DigitalOutput13;
	Cyclic#2.::gHardWare.XP0101Led_1[13] AT %QX."4XP0101.00-00B".DigitalOutput14;
	Cyclic#2.::gHardWare.XP0101Led_1[14] AT %QX."4XP0101.00-00B".DigitalOutput15;
	Cyclic#2.::gHardWare.XP0101Led_1[15] AT %QX."4XP0101.00-00B".DigitalOutput16;
	Cyclic#2.::gHardWare.XP0101Led_1[16] AT %QX."4XP0101.00-00B".DigitalOutput17;
	Cyclic#2.::gHardWare.XP0101Led_1[17] AT %QX."4XP0101.00-00B".DigitalOutput18;
	Cyclic#2.::gHardWare.XP0101Led_1[18] AT %QX."4XP0101.00-00B".DigitalOutput19;
	Cyclic#2.::gHardWare.XP0101Led_1[19] AT %QX."4XP0101.00-00B".DigitalOutput20;
	Cyclic#2.::gHardWare.XP0101Led_1[20] AT %QX."4XP0101.00-00B".DigitalOutput21;
	Cyclic#2.::gHardWare.XP0101Led_1[21] AT %QX."4XP0101.00-00B".DigitalOutput22;
	Cyclic#2.::gHardWare.XP0101Led_1[22] AT %QX."4XP0101.00-00B".DigitalOutput23;
	Cyclic#2.::gHardWare.XP0101Led_1[23] AT %QX."4XP0101.00-00B".DigitalOutput24;
	Cyclic#2.::gHardWare.XP0101Led_1[24] AT %QX."4XP0101.00-00B".DigitalOutput25;
	Cyclic#2.::gHardWare.XP0101Led_1[25] AT %QX."4XP0101.00-00B".DigitalOutput26;
	Cyclic#2.::gHardWare.XP0101Led_1[26] AT %QX."4XP0101.00-00B".DigitalOutput27;
	Cyclic#2.::gHardWare.XP0101Led_1[27] AT %QX."4XP0101.00-00B".DigitalOutput28;
	Cyclic#2.::gHardWare.XP0101Led_1[28] AT %QX."4XP0101.00-00B".DigitalOutput29;
	Cyclic#2.::gHardWare.XP0101Led_1[29] AT %QX."4XP0101.00-00B".DigitalOutput30;
	Cyclic#2.::gHardWare.XP0101Led_1[30] AT %QX."4XP0101.00-00B".DigitalOutput31;
	Cyclic#2.::gHardWare.XP0101Led_1[31] AT %QX."4XP0101.00-00B".DigitalOutput32;
	Cyclic#2.::gExtruderACtrl.InverterStatus.bFault AT %IX."8I84xxxxxxx.01P-1".ETAD_Input_Bool_03;
	Cyclic#2.::gExtruderBCtrl.InverterStatus.bFault AT %IX."8I84xxxxxxx.01P-1a".ETAD_Input_Bool_03;
	Cyclic#2.::gExtruderCCtrl.InverterStatus.bFault AT %IX."8I84xxxxxxx.01P-1b".ETAD_Input_Bool_03;
	::ParisonSacleUp AT %ID."X20DS1119".CounterValue01;
	Cyclic#2.::gAcs380Ctrl.Status.ModuleOk[4] AT %IX."FEPL-02_and_ACS580a1".ModuleOk;
	Cyclic#2.::gAcs380Ctrl.Command.CMDD[4] AT %QW."FEPL-02_and_ACS580a1".ABBCW_I2101Out;
	Cyclic#2.::gAcs380Ctrl.Command.SetSpd[4] AT %QW."FEPL-02_and_ACS580a1".ABBRef1_I2102Out;
	Cyclic#2.::gAcs380Ctrl.Command.SetTor[4] AT %QW."FEPL-02_and_ACS580a1".ABBRef2_I2103Out;
	Cyclic#2.::gAcs380Ctrl.Status.ETAD[4] AT %IW."FEPL-02_and_ACS580a1".ABBSW_I2104;
	Cyclic#2.::gAcs380Ctrl.Status.ActSpd[4] AT %IW."FEPL-02_and_ACS580a1".ABBAct1_I2105;
	Cyclic#2.::gAcs380Ctrl.Status.ActTorque[4] AT %IW."FEPL-02_and_ACS580a1".ABBAct2_I2106;
	Cyclic#2.::gAcs380Ctrl.Status.FaultNum[4] AT %IW."FEPL-02_and_ACS580a1".ErrorCode_I603F;
	Cyclic#2.::gAcs380Ctrl.Status.ActFrequency[4] AT %ID."FEPL-02_and_ACS580a1"._0106_Output_frequency_I4001_S06;
	Cyclic#2.::gAcs380Ctrl.Status.ActCurrent[4] AT %ID."FEPL-02_and_ACS580a1"._0107_Motor_current_I4001_S07;
	Cyclic#2.::gAcs380Ctrl.Status.ActDCVoltage[4] AT %ID."FEPL-02_and_ACS580a1"._0111_DC_voltage_I4001_S0B;
	Cyclic#2.::gAcs380Ctrl.Status.ActPower[4] AT %ID."FEPL-02_and_ACS580a1"._0114_Output_power_I4001_S0E;
	Cyclic#2.::gAcs380Ctrl.Status.ModuleOk[0] AT %IX."FEPL-02_and_ACS580".ModuleOk;
	Cyclic#2.::gAcs380Ctrl.Command.CMDD[0] AT %QW."FEPL-02_and_ACS580".ABBCW_I2101Out;
	Cyclic#2.::gAcs380Ctrl.Command.SetSpd[0] AT %QW."FEPL-02_and_ACS580".ABBRef1_I2102Out;
	Cyclic#2.::gAcs380Ctrl.Command.SetTor[0] AT %QW."FEPL-02_and_ACS580".ABBRef2_I2103Out;
	Cyclic#2.::gAcs380Ctrl.Status.ETAD[0] AT %IW."FEPL-02_and_ACS580".ABBSW_I2104;
	Cyclic#2.::gAcs380Ctrl.Status.ActSpd[0] AT %IW."FEPL-02_and_ACS580".ABBAct1_I2105;
	Cyclic#2.::gAcs380Ctrl.Status.ActTorque[0] AT %IW."FEPL-02_and_ACS580".ABBAct2_I2106;
	Cyclic#2.::gAcs380Ctrl.Status.FaultNum[0] AT %IW."FEPL-02_and_ACS580".ErrorCode_I603F;
	Cyclic#2.::gAcs380Ctrl.Status.ActFrequency[0] AT %ID."FEPL-02_and_ACS580"._0106_Output_frequency_I4001_S06;
	Cyclic#2.::gAcs380Ctrl.Status.ActCurrent[0] AT %ID."FEPL-02_and_ACS580"._0107_Motor_current_I4001_S07;
	Cyclic#2.::gAcs380Ctrl.Status.ActPower[0] AT %ID."FEPL-02_and_ACS580"._0114_Output_power_I4001_S0E;
	Cyclic#2.::gAcs380Ctrl.Status.ModuleOk[3] AT %IX."FEPL-02_and_ACS580a".ModuleOk;
	Cyclic#2.::gAcs380Ctrl.Command.CMDD[3] AT %QW."FEPL-02_and_ACS580a".ABBCW_I2101Out;
	Cyclic#2.::gAcs380Ctrl.Command.SetSpd[3] AT %QW."FEPL-02_and_ACS580a".ABBRef1_I2102Out;
	Cyclic#2.::gAcs380Ctrl.Command.SetTor[3] AT %QW."FEPL-02_and_ACS580a".ABBRef2_I2103Out;
	Cyclic#2.::gAcs380Ctrl.Status.ETAD[3] AT %IW."FEPL-02_and_ACS580a".ABBSW_I2104;
	Cyclic#2.::gAcs380Ctrl.Status.ActSpd[3] AT %IW."FEPL-02_and_ACS580a".ABBAct1_I2105;
	Cyclic#2.::gAcs380Ctrl.Status.ActTorque[3] AT %IW."FEPL-02_and_ACS580a".ABBAct2_I2106;
	Cyclic#2.::gAcs380Ctrl.Status.FaultNum[3] AT %IW."FEPL-02_and_ACS580a".ErrorCode_I603F;
	Cyclic#2.::gAcs380Ctrl.Status.ActDCVoltage[3] AT %ID."FEPL-02_and_ACS580a"._0111_DC_voltage_I4001_S0B;
	Cyclic#2.::gAcs380Ctrl.Status.ActFrequency[3] AT %ID."FEPL-02_and_ACS580a"._0106_Output_frequency_I4001_S06;
	Cyclic#2.::gAcs380Ctrl.Status.ActCurrent[3] AT %ID."FEPL-02_and_ACS580a"._0107_Motor_current_I4001_S07;
	Cyclic#2.::gAcs380Ctrl.Status.ActPower[3] AT %ID."FEPL-02_and_ACS580a"._0114_Output_power_I4001_S0E;
	::gHardWare.ModuleOk.PS3300_2 AT %IX."X20PS3300a".ModuleOk;
	Cyclic#2.::gHardWare.ModuleOk.AI4632_3 AT %IX."X20AI4632_C".ModuleOk;
	Cyclic#1.::gHardWare.AI4632_3[0] AT %IW."X20AI4632_C".AnalogInput01;
	Cyclic#1.::gHardWare.AI4632_3[1] AT %IW."X20AI4632_C".AnalogInput02;
	Cyclic#1.::gHardWare.AI4632_3[2] AT %IW."X20AI4632_C".AnalogInput03;
	Cyclic#1.::gHardWare.AI4632_3[3] AT %IW."X20AI4632_C".AnalogInput04;
	Cyclic#2.::gAcs380Ctrl.Status.ModuleOk[1] AT %IX."FEPL-02_and_ACS580a2".ModuleOk;
	Cyclic#2.::gAcs380Ctrl.Command.CMDD[1] AT %QW."FEPL-02_and_ACS580a2".ABBCW_I2101Out;
	Cyclic#2.::gAcs380Ctrl.Command.SetSpd[1] AT %QW."FEPL-02_and_ACS580a2".ABBRef1_I2102Out;
	Cyclic#2.::gAcs380Ctrl.Command.SetTor[1] AT %QW."FEPL-02_and_ACS580a2".ABBRef2_I2103Out;
	Cyclic#2.::gAcs380Ctrl.Status.ETAD[1] AT %IW."FEPL-02_and_ACS580a2".ABBSW_I2104;
	Cyclic#2.::gAcs380Ctrl.Status.ActSpd[1] AT %IW."FEPL-02_and_ACS580a2".ABBAct1_I2105;
	Cyclic#2.::gAcs380Ctrl.Status.ActTorque[1] AT %IW."FEPL-02_and_ACS580a2".ABBAct2_I2106;
	Cyclic#2.::gAcs380Ctrl.Status.FaultNum[1] AT %IW."FEPL-02_and_ACS580a2".ErrorCode_I603F;
	Cyclic#2.::gAcs380Ctrl.Status.ActFrequency[1] AT %ID."FEPL-02_and_ACS580a2"._0106_Output_frequency_I4001_S06;
	Cyclic#2.::gAcs380Ctrl.Status.ActCurrent[1] AT %ID."FEPL-02_and_ACS580a2"._0107_Motor_current_I4001_S07;
	Cyclic#2.::gAcs380Ctrl.Status.ActDCVoltage[1] AT %ID."FEPL-02_and_ACS580a2"._0111_DC_voltage_I4001_S0B;
	Cyclic#2.::gAcs380Ctrl.Status.ActPower[1] AT %ID."FEPL-02_and_ACS580a2"._0114_Output_power_I4001_S0E;
	Cyclic#2.::gAcs380Ctrl.Status.ModuleOk[2] AT %IX."FEPL-02_and_ACS580a2a".ModuleOk;
	Cyclic#2.::gAcs380Ctrl.Command.CMDD[2] AT %QW."FEPL-02_and_ACS580a2a".ABBCW_I2101Out;
	Cyclic#2.::gAcs380Ctrl.Command.SetSpd[2] AT %QW."FEPL-02_and_ACS580a2a".ABBRef1_I2102Out;
	Cyclic#2.::gAcs380Ctrl.Command.SetTor[2] AT %QW."FEPL-02_and_ACS580a2a".ABBRef2_I2103Out;
	Cyclic#2.::gAcs380Ctrl.Status.ETAD[2] AT %IW."FEPL-02_and_ACS580a2a".ABBSW_I2104;
	Cyclic#2.::gAcs380Ctrl.Status.ActSpd[2] AT %IW."FEPL-02_and_ACS580a2a".ABBAct1_I2105;
	Cyclic#2.::gAcs380Ctrl.Status.ActTorque[2] AT %IW."FEPL-02_and_ACS580a2a".ABBAct2_I2106;
	Cyclic#2.::gAcs380Ctrl.Status.FaultNum[2] AT %IW."FEPL-02_and_ACS580a2a".ErrorCode_I603F;
	Cyclic#2.::gAcs380Ctrl.Status.ActFrequency[2] AT %ID."FEPL-02_and_ACS580a2a"._0106_Output_frequency_I4001_S06;
	Cyclic#2.::gAcs380Ctrl.Status.ActDCVoltage[0] AT %ID."FEPL-02_and_ACS580"._0111_DC_voltage_I4001_S0B;
	Cyclic#2.::gAcs380Ctrl.Status.ActCurrent[2] AT %ID."FEPL-02_and_ACS580a2a"._0107_Motor_current_I4001_S07;
	Cyclic#2.::gAcs380Ctrl.Status.ActDCVoltage[2] AT %ID."FEPL-02_and_ACS580a2a"._0111_DC_voltage_I4001_S0B;
	Cyclic#2.::gAcs380Ctrl.Status.ActPower[2] AT %ID."FEPL-02_and_ACS580a2a"._0114_Output_power_I4001_S0E;
	Cyclic#1.::gHardWare.AO4632_1[0] AT %QW."X20AO4632_A".AnalogOutput01;
	Cyclic#1.::gHardWare.AO4632_1[1] AT %QW."X20AO4632_A".AnalogOutput02;
	Cyclic#1.::gHardWare.AO4632_1[2] AT %QW."X20AO4632_A".AnalogOutput03;
	Cyclic#1.::gHardWare.AO4632_1[3] AT %QW."X20AO4632_A".AnalogOutput04;
	Cyclic#1.::gHardWare.ModuleOk.AO4632_1 AT %IX."X20AO4632_A".ModuleOk;
	::gHardWare.ModuleOk.BC0083_1 AT %IX."X20BC0083".ModuleOk;
	::gHardWare.ModuleOk.PS9400_1 AT %IX."X20PS9400".ModuleOk;
	Cyclic#1.::gHardWare.ModuleOk.AO4632_2 AT %IX."X20AO4632_B".ModuleOk;
	Cyclic#1.::gHardWare.AO4632_2[0] AT %QW."X20AO4632_B".AnalogOutput01;
	Cyclic#1.::gHardWare.AO4632_2[1] AT %QW."X20AO4632_B".AnalogOutput02;
	Cyclic#1.::gHardWare.AO4632_2[2] AT %QW."X20AO4632_B".AnalogOutput03;
	Cyclic#1.::gHardWare.AO4632_2[3] AT %QW."X20AO4632_B".AnalogOutput04;
	Cyclic#1.::gHardWare.ModuleOk.AO4632_3 AT %IX."X20AO4632_C".ModuleOk;
	Cyclic#1.::gHardWare.AO4632_3[0] AT %QW."X20AO4632_C".AnalogOutput01;
	Cyclic#1.::gHardWare.AO4632_3[1] AT %QW."X20AO4632_C".AnalogOutput02;
	Cyclic#1.::gHardWare.AO4632_3[2] AT %QW."X20AO4632_C".AnalogOutput03;
	Cyclic#1.::gHardWare.AO4632_3[3] AT %QW."X20AO4632_C".AnalogOutput04;
	Cyclic#1.::gHardWare.ModuleOk.AO4632_4 AT %IX."X20AO4632_D".ModuleOk;
	Cyclic#1.::gHardWare.AO4632_4[0] AT %QW."X20AO4632_D".AnalogOutput01;
	Cyclic#1.::gHardWare.AO4632_4[1] AT %QW."X20AO4632_D".AnalogOutput02;
	Cyclic#1.::gHardWare.AO4632_4[2] AT %QW."X20AO4632_D".AnalogOutput03;
	Cyclic#1.::gHardWare.AO4632_4[3] AT %QW."X20AO4632_D".AnalogOutput04;
	::gHardWare.ModuleOk.BC0083_2  AT %IX."X20BC0083b".ModuleOk;
	::gHardWare.ModuleOk.PS9400_2  AT %IX."X20PS9400b".ModuleOk;
END_VAR
```

### Acp10cfg.ncc - 5PPC2100_BY01_000/Motion/Acp10cfg.ncc
```
NcConfiguration (Version=2.48.1, NcSwId=Acp10)
  ACP10CF1_typ:
    cnt_nettrc_rec_drive = 150
    bufsize_trace_upload = 1200
    tc_nc_man_task = Cyclic #1
    glob_pv_as_ncobject = Yes
    ncsys_dl_broadcast = Yes
    ncsys_dl_acp_reset = Yes
    safemc_log_err_to_ax = Yes
    network_init:
      ncsw_init_execute = Yes
      automatic_execute = No
      node_nr_warning = Yes
      net_err_before_ncact = Yes
    nettrc:
      enter_parsecrec = Yes
      enter_ncaction = Yes
      save_ring_startidx = No
    cam_prof_download:
      cam_dat_dl_parallel = No
      tc_cam_dl_parallel = Task class for NC Manager task
    plk_if[0]:
      if_name = SL1.IF1
      tc_CycDat_PLCopen = Task class for NC Manager task
      mc_broadcast_extdat = No
```
